LIN {X 0,Y 541.507,Z 325.44,A -85,B 0,C 180,E1 25518.834,E2 25518.834} C_VEL
LIN {X 0,Y 542.9,Z 340.233,A -85,B 0,C 180,E1 25517.69,E2 25517.69} C_VEL
LIN {X 0,Y 545.785,Z 352.594,A -85,B 0,C 180,E1 25516.608,E2 25516.608} C_VEL
LIN {X 0,Y 549.602,Z 361.822,A -85,B 0,C 180,E1 25515.687,E2 25515.687} C_VEL
LIN {X 0,Y 554.796,Z 369.914,A -85,B 0,C 180,E1 25514.76,E2 25514.76} C_VEL
LIN {X 0,Y 561.405,Z 376.773,A -85,B 0,C 180,E1 25513.838,E2 25513.838} C_VEL
LIN {X 0,Y 569.472,Z 382.283,A -85,B 0,C 180,E1 25512.933,E2 25512.933} C_VEL
LIN {X 0,Y 575.782,Z 385.075,A -85,B 0,C 180,E1 25512.29,E2 25512.29} C_VEL
LIN {X 0,Y 579.36,Z 385.747,A -85,B 0,C 180,E1 25511.772,E2 25511.772} C_VEL
LIN {X 0,Y 581.974,Z 385.283,A -85,B 0,C 180,E1 25511.193,E2 25511.193} C_VEL
LIN {X 0,Y 583.328,Z 383.79,A -85,B 0,C 180,E1 25510.595,E2 25510.595} C_VEL
LIN {X 0,Y 583.299,Z 381.198,A -85,B 0,C 180,E1 25509.985,E2 25509.985} C_VEL
LIN {X 0,Y 581.736,Z 377.706,A -85,B 0,C 180,E1 25509.426,E2 25509.426} C_VEL
LIN {X 0,Y 578.601,Z 373.318,A -85,B 0,C 180,E1 25508.946,E2 25508.946} C_VEL
LIN {X 0,Y 572.524,Z 363.934,A -85,B 0,C 180,E1 25508.187,E2 25508.187} C_VEL
LIN {X 0,Y 567.538,Z 353.434,A -85,B 0,C 180,E1 25507.542,E2 25507.542} C_VEL
LIN {X 0,Y 563.487,Z 341.539,A -85,B 0,C 180,E1 25507.003,E2 25507.003} C_VEL
LIN {X 0,Y 562.249,Z 337.195,A -85,B 0,C 180,E1 25506.836,E2 25506.836} C_VEL
LIN {X 0,Y 557.951,Z 382.113,A -85,B 0,C 180,E1 25506.242,E2 25506.242} C_VEL
LIN {X 0,Y 554.59,Z 408.363,A -85,B 0,C 180,E1 25505.766,E2 25505.766} C_VEL
LIN {X 0,Y 552.443,Z 419.215,A -85,B 0,C 180,E1 25505.456,E2 25505.456} C_VEL
LIN {X 0,Y 551.439,Z 422.72,A -85,B 0,C 180,E1 25505.309,E2 25505.309} C_VEL
LIN {X 0,Y 547.112,Z 475.176,A -85,B 0,C 180,E1 25504.664,E2 25504.664} C_VEL
LIN {X 0,Y 544.575,Z 495.316,A -85,B 0,C 180,E1 25504.346,E2 25504.346} C_VEL
LIN {X 0,Y 541.642,Z 509.391,A -85,B 0,C 180,E1 25504.002,E2 25504.002} C_VEL
LIN {X 0,Y 539.647,Z 516.391,A -85,B 0,C 180,E1 25503.689,E2 25503.689} C_VEL
LIN {X 0,Y 538.533,Z 609.219,A -85,B 0,C 180,E1 25502.262,E2 25502.262} C_VEL
LIN {X 0,Y 537.892,Z 631.012,A -85,B 0,C 180,E1 25501.735,E2 25501.735} C_VEL
LIN {X 0,Y 537.114,Z 653.311,A -85,B 0,C 180,E1 25500.979,E2 25500.979} C_VEL
LIN {X 0,Y 536.157,Z 674.428,A -85,B 0,C 180,E1 25500.054,E2 25500.054} C_VEL
LIN {X 0,Y 535.132,Z 694.792,A -85,B 0,C 180,E1 25498.942,E2 25498.942} C_VEL
LIN {X 0,Y 534.004,Z 714.986,A -85,B 0,C 180,E1 25497.608,E2 25497.608} C_VEL
LIN {X 0,Y 532.851,Z 734.82,A -85,B 0,C 180,E1 25496.046,E2 25496.046} C_VEL
LIN {X 0,Y 531.811,Z 752.831,A -85,B 0,C 180,E1 25494.374,E2 25494.374} C_VEL
LIN {X 0,Y 530.82,Z 770.22,A -85,B 0,C 180,E1 25492.481,E2 25492.481} C_VEL
LIN {X 0,Y 529.957,Z 786.287,A -85,B 0,C 180,E1 25490.428,E2 25490.428} C_VEL
LIN {X 0,Y 529.266,Z 800.604,A -85,B 0,C 180,E1 25488.276,E2 25488.276} C_VEL
LIN {X 0,Y 528.733,Z 813.274,A -85,B 0,C 180,E1 25486.027,E2 25486.027} C_VEL
LIN {X 0,Y 528.362,Z 824.318,A -85,B 0,C 180,E1 25483.683,E2 25483.683} C_VEL
LIN {X 0,Y 528.131,Z 833.313,A -85,B 0,C 180,E1 25481.355,E2 25481.355} C_VEL
LIN {X 0,Y 528.003,Z 840.399,A -85,B 0,C 180,E1 25479.043,E2 25479.043} C_VEL
LIN {X 0,Y 527.934,Z 846.011,A -85,B 0,C 180,E1 25476.634,E2 25476.634} C_VEL
LIN {X 0,Y 527.917,Z 849.739,A -85,B 0,C 180,E1 25474.345,E2 25474.345} C_VEL
LIN {X 0,Y 527.909,Z 851.902,A -85,B 0,C 180,E1 25471.954,E2 25471.954} C_VEL
LIN {X 0,Y 527.898,Z 852.445,A -85,B 0,C 180,E1 25469.566,E2 25469.566} C_VEL
LIN {X 0,Y 527.91,Z 851.331,A -85,B 0,C 180,E1 25467.177,E2 25467.177} C_VEL
LIN {X 0,Y 527.923,Z 848.489,A -85,B 0,C 180,E1 25464.784,E2 25464.784} C_VEL
LIN {X 0,Y 527.955,Z 843.939,A -85,B 0,C 180,E1 25462.382,E2 25462.382} C_VEL
LIN {X 0,Y 528.035,Z 837.923,A -85,B 0,C 180,E1 25460.078,E2 25460.078} C_VEL
LIN {X 0,Y 528.2,Z 830.099,A -85,B 0,C 180,E1 25457.76,E2 25457.76} C_VEL
LIN {X 0,Y 528.485,Z 820.356,A -85,B 0,C 180,E1 25455.426,E2 25455.426} C_VEL
LIN {X 0,Y 528.903,Z 809.121,A -85,B 0,C 180,E1 25453.188,E2 25453.188} C_VEL
LIN {X 0,Y 529.496,Z 795.627,A -85,B 0,C 180,E1 25450.932,E2 25450.932} C_VEL
LIN {X 0,Y 530.266,Z 780.344,A -85,B 0,C 180,E1 25448.775,E2 25448.775} C_VEL
LIN {X 0,Y 531.183,Z 763.692,A -85,B 0,C 180,E1 25446.774,E2 25446.774} C_VEL
LIN {X 0,Y 532.215,Z 745.663,A -85,B 0,C 180,E1 25444.929,E2 25444.929} C_VEL
LIN {X 0,Y 533.303,Z 727.139,A -85,B 0,C 180,E1 25443.319,E2 25443.319} C_VEL
LIN {X 0,Y 534.441,Z 707.515,A -85,B 0,C 180,E1 25441.871,E2 25441.871} C_VEL
LIN {X 0,Y 535.472,Z 687.857,A -85,B 0,C 180,E1 25440.655,E2 25440.655} C_VEL
LIN {X 0,Y 536.509,Z 667.145,A -85,B 0,C 180,E1 25439.603,E2 25439.603} C_VEL
LIN {X 0,Y 537.398,Z 645.684,A -85,B 0,C 180,E1 25438.736,E2 25438.736} C_VEL
LIN {X 0,Y 538.141,Z 623.996,A -85,B 0,C 180,E1 25438.074,E2 25438.074} C_VEL
LIN {X 0,Y 538.654,Z 601.949,A -85,B 0,C 180,E1 25437.607,E2 25437.607} C_VEL
LIN {X 0,Y 539.603,Z 521.674,A -85,B 0,C 180,E1 25436.387,E2 25436.387} C_VEL
LIN {X 0,Y 541.451,Z 515.855,A -85,B 0,C 180,E1 25436.104,E2 25436.104} C_VEL
LIN {X 0,Y 544.043,Z 503.404,A -85,B 0,C 180,E1 25435.787,E2 25435.787} C_VEL
LIN {X 0,Y 547.469,Z 471.343,A -85,B 0,C 180,E1 25435.282,E2 25435.282} C_VEL
LIN {X 0,Y 551.647,Z 421.541,A -85,B 0,C 180,E1 25434.661,E2 25434.661} C_VEL
LIN {X 0,Y 553.46,Z 414.673,A -85,B 0,C 180,E1 25434.397,E2 25434.397} C_VEL
LIN {X 0,Y 556.22,Z 396.703,A -85,B 0,C 180,E1 25434.002,E2 25434.002} C_VEL
LIN {X 0,Y 559.935,Z 363.496,A -85,B 0,C 180,E1 25433.482,E2 25433.482} C_VEL
LIN {X 0,Y 562.811,Z 376.767,A -85,B 0,C 180,E1 25433.088,E2 25433.088} C_VEL
LIN {X 0,Y 566.701,Z 388.825,A -85,B 0,C 180,E1 25432.568,E2 25432.568} C_VEL
LIN {X 0,Y 571.599,Z 399.681,A -85,B 0,C 180,E1 25431.931,E2 25431.931} C_VEL
LIN {X 0,Y 577.324,Z 409.005,A -85,B 0,C 180,E1 25431.206,E2 25431.206} C_VEL
LIN {X 0,Y 579.654,Z 413.297,A -85,B 0,C 180,E1 25430.724,E2 25430.724} C_VEL
LIN {X 0,Y 580.529,Z 416.774,A -85,B 0,C 180,E1 25430.155,E2 25430.155} C_VEL
LIN {X 0,Y 580.022,Z 419.104,A -85,B 0,C 180,E1 25429.597,E2 25429.597} C_VEL
LIN {X 0,Y 578.027,Z 420.583,A -85,B 0,C 180,E1 25428.954,E2 25428.954} C_VEL
LIN {X 0,Y 574.752,Z 420.735,A -85,B 0,C 180,E1 25428.352,E2 25428.352} C_VEL
LIN {X 0,Y 570.602,Z 419.567,A -85,B 0,C 180,E1 25427.835,E2 25427.835} C_VEL
LIN {X 0,Y 562.188,Z 414.887,A -85,B 0,C 180,E1 25426.967,E2 25426.967} C_VEL
LIN {X 0,Y 554.609,Z 408.372,A -85,B 0,C 180,E1 25425.998,E2 25425.998} C_VEL
LIN {X 0,Y 548.567,Z 400.431,A -85,B 0,C 180,E1 25424.992,E2 25424.992} C_VEL
LIN {X 0,Y 543.999,Z 390.85,A -85,B 0,C 180,E1 25423.934,E2 25423.934} C_VEL
LIN {X 0,Y 540.909,Z 379.13,A -85,B 0,C 180,E1 25422.79,E2 25422.79} C_VEL
LIN {X 0,Y 539.455,Z 365.314,A -85,B 0,C 180,E1 25421.57,E2 25421.57} C_VEL
LIN {X 0,Y 540.181,Z 339.074,A -85,B 0,C 180,E1 25419.479,E2 25419.479} C_VEL
LIN {X 0,Y 542.247,Z 299.859,A -85,B 0,C 180,E1 25416.312,E2 25416.312} C_VEL
LIN {X 0,Y 543.435,Z 278.465,A -85,B 0,C 180,E1 25414.519,E2 25414.519} C_VEL
LIN {X 0,Y 536.159,Z 263.024,A -85,B 0,C 180,E1 25412.232,E2 25412.232} C_VEL
LIN {X 0,Y 532.304,Z 255.135,A -85,B 0,C 180,E1 25410.975,E2 25410.975} C_VEL
LIN {X 0,Y 530.079,Z 250.727,A -85,B 0,C 180,E1 25410.24,E2 25410.24} C_VEL
LIN {X 0,Y 528.598,Z 247.484,A -85,B 0,C 180,E1 25409.708,E2 25409.708} C_VEL
LIN {X 0,Y 528.503,Z 246.905,A -85,B 0,C 180,E1 25409.589,E2 25409.589} C_VEL
LIN {X 0,Y 528.518,Z 247.111,A -85,B 0,C 180,E1 25407.776,E2 25407.776} C_VEL
LIN {X 0,Y 530.21,Z 254.424,A -85,B 0,C 180,E1 25407.274,E2 25407.274} C_VEL
LIN {X 0,Y 530.852,Z 299.671,A -85,B 0,C 180,E1 25404.42,E2 25404.42} C_VEL
LIN {X 0,Y 531.29,Z 341.245,A -85,B 0,C 180,E1 25401.645,E2 25401.645} C_VEL
LIN {X 0,Y 531.277,Z 383.369,A -85,B 0,C 180,E1 25398.716,E2 25398.716} C_VEL
LIN {X 0,Y 530.854,Z 431.931,A -85,B 0,C 180,E1 25395.233,E2 25395.233} C_VEL
LIN {X 0,Y 530.24,Z 479.348,A -85,B 0,C 180,E1 25391.75,E2 25391.75} C_VEL
LIN {X 0,Y 530.109,Z 491.534,A -85,B 0,C 180,E1 25390.885,E2 25390.885} C_VEL
LIN {X 0,Y 529.689,Z 604.749,A -85,B 0,C 180,E1 25389.291,E2 25389.291} C_VEL
LIN {X 0,Y 529.568,Z 619.615,A -85,B 0,C 180,E1 25388.872,E2 25388.872} C_VEL
LIN {X 0,Y 529.421,Z 632.902,A -85,B 0,C 180,E1 25388.307,E2 25388.307} C_VEL
LIN {X 0,Y 529.2,Z 645.983,A -85,B 0,C 180,E1 25387.545,E2 25387.545} C_VEL
LIN {X 0,Y 528.96,Z 658.621,A -85,B 0,C 180,E1 25386.566,E2 25386.566} C_VEL
LIN {X 0,Y 528.737,Z 669.029,A -85,B 0,C 180,E1 25385.534,E2 25385.534} C_VEL
LIN {X 0,Y 528.525,Z 678.575,A -85,B 0,C 180,E1 25384.339,E2 25384.339} C_VEL
LIN {X 0,Y 528.346,Z 687.273,A -85,B 0,C 180,E1 25382.928,E2 25382.928} C_VEL
LIN {X 0,Y 528.206,Z 693.851,A -85,B 0,C 180,E1 25381.518,E2 25381.518} C_VEL
LIN {X 0,Y 528.13,Z 699.006,A -85,B 0,C 180,E1 25380,E2 25380} C_VEL
LIN {X 0,Y 528.078,Z 702.566,A -85,B 0,C 180,E1 25378.372,E2 25378.372} C_VEL
LIN {X 0,Y 528.064,Z 704.318,A -85,B 0,C 180,E1 25376.635,E2 25376.635} C_VEL
LIN {X 0,Y 528.051,Z 704.126,A -85,B 0,C 180,E1 25375.003,E2 25375.003} C_VEL
LIN {X 0,Y 528.068,Z 702.145,A -85,B 0,C 180,E1 25373.367,E2 25373.367} C_VEL
LIN {X 0,Y 528.104,Z 698.628,A -85,B 0,C 180,E1 25371.836,E2 25371.836} C_VEL
LIN {X 0,Y 528.191,Z 692.798,A -85,B 0,C 180,E1 25370.19,E2 25370.19} C_VEL
LIN {X 0,Y 528.319,Z 685.733,A -85,B 0,C 180,E1 25368.759,E2 25368.759} C_VEL
LIN {X 0,Y 528.492,Z 677.206,A -85,B 0,C 180,E1 25367.433,E2 25367.433} C_VEL
LIN {X 0,Y 528.72,Z 667.179,A -85,B 0,C 180,E1 25366.215,E2 25366.215} C_VEL
LIN {X 0,Y 528.965,Z 655.414,A -85,B 0,C 180,E1 25365.103,E2 25365.103} C_VEL
LIN {X 0,Y 529.203,Z 643.22,A -85,B 0,C 180,E1 25364.212,E2 25364.212} C_VEL
LIN {X 0,Y 529.426,Z 630.244,A -85,B 0,C 180,E1 25363.487,E2 25363.487} C_VEL
LIN {X 0,Y 529.616,Z 615.198,A -85,B 0,C 180,E1 25362.889,E2 25362.889} C_VEL
LIN {X 0,Y 529.731,Z 599.229,A -85,B 0,C 180,E1 25362.502,E2 25362.502} C_VEL
LIN {X 0,Y 529.967,Z 489.753,A -85,B 0,C 180,E1 25360.978,E2 25360.978} C_VEL
LIN {X 0,Y 529.944,Z 486.878,A -85,B 0,C 180,E1 25360.802,E2 25360.802} C_VEL
LIN {X 0,Y 530.358,Z 460.271,A -85,B 0,C 180,E1 25358.814,E2 25358.814} C_VEL
LIN {X 0,Y 529.49,Z 454.16,A -85,B 0,C 180,E1 25358.319,E2 25358.319} C_VEL
LIN {X 0,Y 523.776,Z 438.358,A -85,B 0,C 180,E1 25356.901,E2 25356.901} C_VEL
LIN {X 0,Y 523.166,Z 432.941,A -85,B 0,C 180,E1 25356.467,E2 25356.467} C_VEL
LIN {X 0,Y 523.904,Z 387.135,A -85,B 0,C 180,E1 25353.033,E2 25353.033} C_VEL
LIN {X 0,Y 524.522,Z 341.101,A -85,B 0,C 180,E1 25349.595,E2 25349.595} C_VEL
LIN {X 0,Y 524.914,Z 297.566,A -85,B 0,C 180,E1 25346.337,E2 25346.337} C_VEL
LIN {X 0,Y 525.147,Z 262.725,A -85,B 0,C 180,E1 25343.739,E2 25343.739} C_VEL
LIN {X 0,Y 520.574,Z 247.885,A -85,B 0,C 180,E1 25342.354,E2 25342.354} C_VEL
LIN {X 0,Y 520.575,Z 247.892,A -85,B 0,C 180,E1 25338.791,E2 25338.791} C_VEL
LIN {X 0,Y 520.564,Z 247.895,A -85,B 0,C 180,E1 25335.446,E2 25335.446} C_VEL
LIN {X 0,Y 520.591,Z 247.964,A -85,B 0,C 180,E1 25333.248,E2 25333.248} C_VEL
LIN {X 0,Y 521.88,Z 251.385,A -85,B 0,C 180,E1 25332.633,E2 25332.633} C_VEL
LIN {X 0,Y 524.834,Z 257.768,A -85,B 0,C 180,E1 25331.439,E2 25331.439} C_VEL
LIN {X 0,Y 530.138,Z 269.708,A -85,B 0,C 180,E1 25329.325,E2 25329.325} C_VEL
LIN {X 0,Y 532.076,Z 275.112,A -85,B 0,C 180,E1 25328.463,E2 25328.463} C_VEL
LIN {X 0,Y 529.458,Z 306.929,A -85,B 0,C 180,E1 25325.183,E2 25325.183} C_VEL
LIN {X 0,Y 531.569,Z 317.62,A -85,B 0,C 180,E1 25324.852,E2 25324.852} C_VEL
LIN {X 0,Y 528.989,Z 544.595,A -85,B 0,C 180,E1 25321.435,E2 25321.435} C_VEL
LIN {X 0,Y 528.578,Z 567.627,A -85,B 0,C 180,E1 25321.026,E2 25321.026} C_VEL
LIN {X 0,Y 527.977,Z 588.155,A -85,B 0,C 180,E1 25320.456,E2 25320.456} C_VEL
LIN {X 0,Y 527.322,Z 605.247,A -85,B 0,C 180,E1 25319.819,E2 25319.819} C_VEL
LIN {X 0,Y 526.551,Z 623.634,A -85,B 0,C 180,E1 25318.961,E2 25318.961} C_VEL
LIN {X 0,Y 525.565,Z 642.685,A -85,B 0,C 180,E1 25317.843,E2 25317.843} C_VEL
LIN {X 0,Y 524.73,Z 658.626,A -85,B 0,C 180,E1 25316.724,E2 25316.724} C_VEL
LIN {X 0,Y 523.753,Z 676.293,A -85,B 0,C 180,E1 25315.257,E2 25315.257} C_VEL
LIN {X 0,Y 522.9,Z 691.093,A -85,B 0,C 180,E1 25313.795,E2 25313.795} C_VEL
LIN {X 0,Y 522.144,Z 705.392,A -85,B 0,C 180,E1 25312.163,E2 25312.163} C_VEL
LIN {X 0,Y 521.439,Z 719.102,A -85,B 0,C 180,E1 25310.308,E2 25310.308} C_VEL
LIN {X 0,Y 520.919,Z 730.743,A -85,B 0,C 180,E1 25308.464,E2 25308.464} C_VEL
LIN {X 0,Y 520.481,Z 742.217,A -85,B 0,C 180,E1 25306.288,E2 25306.288} C_VEL
LIN {X 0,Y 520.219,Z 750.632,A -85,B 0,C 180,E1 25304.356,E2 25304.356} C_VEL
LIN {X 0,Y 520.054,Z 758.283,A -85,B 0,C 180,E1 25302.21,E2 25302.21} C_VEL
LIN {X 0,Y 519.961,Z 764.345,A -85,B 0,C 180,E1 25299.966,E2 25299.966} C_VEL
LIN {X 0,Y 519.929,Z 768.375,A -85,B 0,C 180,E1 25297.95,E2 25297.95} C_VEL
LIN {X 0,Y 519.907,Z 771.321,A -85,B 0,C 180,E1 25295.629,E2 25295.629} C_VEL
LIN {X 0,Y 519.903,Z 772.378,A -85,B 0,C 180,E1 25293.503,E2 25293.503} C_VEL
LIN {X 0,Y 519.903,Z 772.051,A -85,B 0,C 180,E1 25291.322,E2 25291.322} C_VEL
LIN {X 0,Y 519.918,Z 769.904,A -85,B 0,C 180,E1 25289.008,E2 25289.008} C_VEL
LIN {X 0,Y 519.938,Z 766.672,A -85,B 0,C 180,E1 25287.024,E2 25287.024} C_VEL
LIN {X 0,Y 519.998,Z 761.549,A -85,B 0,C 180,E1 25284.815,E2 25284.815} C_VEL
LIN {X 0,Y 520.128,Z 754.549,A -85,B 0,C 180,E1 25282.6,E2 25282.6} C_VEL
LIN {X 0,Y 520.317,Z 747.153,A -85,B 0,C 180,E1 25280.711,E2 25280.711} C_VEL
LIN {X 0,Y 520.674,Z 737.117,A -85,B 0,C 180,E1 25278.592,E2 25278.592} C_VEL
LIN {X 0,Y 521.109,Z 726.154,A -85,B 0,C 180,E1 25276.688,E2 25276.688} C_VEL
LIN {X 0,Y 521.687,Z 714.146,A -85,B 0,C 180,E1 25274.891,E2 25274.891} C_VEL
LIN {X 0,Y 522.451,Z 699.354,A -85,B 0,C 180,E1 25273.031,E2 25273.031} C_VEL
LIN {X 0,Y 523.195,Z 685.995,A -85,B 0,C 180,E1 25271.588,E2 25271.588} C_VEL
LIN {X 0,Y 524.155,Z 669.279,A -85,B 0,C 180,E1 25270.034,E2 25270.034} C_VEL
LIN {X 0,Y 525.053,Z 652.42,A -85,B 0,C 180,E1 25268.729,E2 25268.729} C_VEL
LIN {X 0,Y 525.934,Z 636.075,A -85,B 0,C 180,E1 25267.652,E2 25267.652} C_VEL
LIN {X 0,Y 526.869,Z 616.032,A -85,B 0,C 180,E1 25266.573,E2 25266.573} C_VEL
LIN {X 0,Y 527.585,Z 598.852,A -85,B 0,C 180,E1 25265.836,E2 25265.836} C_VEL
LIN {X 0,Y 528.241,Z 580.125,A -85,B 0,C 180,E1 25265.201,E2 25265.201} C_VEL
LIN {X 0,Y 528.768,Z 559.287,A -85,B 0,C 180,E1 25264.715,E2 25264.715} C_VEL
LIN {X 0,Y 531.644,Z 314.439,A -85,B 0,C 180,E1 25261.011,E2 25261.011} C_VEL
LIN {X 0,Y 529.934,Z 304.934,A -85,B 0,C 180,E1 25260.716,E2 25260.716} C_VEL
LIN {X 0,Y 532.112,Z 274.325,A -85,B 0,C 180,E1 25258.065,E2 25258.065} C_VEL
LIN {X 0,Y 529.618,Z 267.665,A -85,B 0,C 180,E1 25257.153,E2 25257.153} C_VEL
LIN {X 0,Y 523.77,Z 255.31,A -85,B 0,C 180,E1 25255.267,E2 25255.267} C_VEL
LIN {X 0,Y 522.007,Z 251.554,A -85,B 0,C 180,E1 25254.684,E2 25254.684} C_VEL
LIN {X 0,Y 520.594,Z 247.941,A -85,B 0,C 180,E1 25254.153,E2 25254.153} C_VEL
LIN {X 0,Y 520.583,Z 247.897,A -85,B 0,C 180,E1 25250.667,E2 25250.667} C_VEL
LIN {X 0,Y 520.576,Z 247.893,A -85,B 0,C 180,E1 25247.162,E2 25247.162} C_VEL
LIN {X 0,Y 520.585,Z 247.89,A -85,B 0,C 180,E1 25243.592,E2 25243.592} C_VEL
LIN {X 0,Y 520.589,Z 247.883,A -85,B 0,C 180,E1 25239.974,E2 25239.974} C_VEL
LIN {X 0,Y 520.57,Z 247.88,A -85,B 0,C 180,E1 25236.543,E2 25236.543} C_VEL
LIN {X 0,Y 520.567,Z 247.893,A -85,B 0,C 180,E1 25233.13,E2 25233.13} C_VEL
LIN {X 0,Y 520.582,Z 247.891,A -85,B 0,C 180,E1 25229.705,E2 25229.705} C_VEL
LIN {X 0,Y 520.591,Z 247.925,A -85,B 0,C 180,E1 25229.168,E2 25229.168} C_VEL
LIN {X 0,Y 525.449,Z 263.917,A -85,B 0,C 180,E1 25227.604,E2 25227.604} C_VEL
LIN {X 0,Y 525.069,Z 309.421,A -85,B 0,C 180,E1 25223.929,E2 25223.929} C_VEL
LIN {X 0,Y 524.544,Z 350.281,A -85,B 0,C 180,E1 25220.622,E2 25220.622} C_VEL
LIN {X 0,Y 523.837,Z 391.693,A -85,B 0,C 180,E1 25217.266,E2 25217.266} C_VEL
LIN {X 0,Y 523.058,Z 434.806,A -85,B 0,C 180,E1 25213.774,E2 25213.774} C_VEL
LIN {X 0,Y 523.011,Z 441.178,A -85,B 0,C 180,E1 25213.284,E2 25213.284} C_VEL
LIN {X 0,Y 523.43,Z 448.653,A -85,B 0,C 180,E1 25213.159,E2 25213.159} C_VEL
LIN {X 0,Y 522.655,Z 583.279,A -85,B 0,C 180,E1 25211.221,E2 25211.221} C_VEL
LIN {X 0,Y 522.498,Z 600.137,A -85,B 0,C 180,E1 25210.764,E2 25210.764} C_VEL
LIN {X 0,Y 522.241,Z 615.223,A -85,B 0,C 180,E1 25210.145,E2 25210.145} C_VEL
LIN {X 0,Y 521.93,Z 630.251,A -85,B 0,C 180,E1 25209.316,E2 25209.316} C_VEL
LIN {X 0,Y 521.561,Z 643.994,A -85,B 0,C 180,E1 25208.322,E2 25208.322} C_VEL
LIN {X 0,Y 521.215,Z 656.762,A -85,B 0,C 180,E1 25207.163,E2 25207.163} C_VEL
LIN {X 0,Y 520.87,Z 668.3,A -85,B 0,C 180,E1 25205.84,E2 25205.84} C_VEL
LIN {X 0,Y 520.592,Z 678.338,A -85,B 0,C 180,E1 25204.406,E2 25204.406} C_VEL
LIN {X 0,Y 520.364,Z 687.336,A -85,B 0,C 180,E1 25202.754,E2 25202.754} C_VEL
LIN {X 0,Y 520.235,Z 694.19,A -85,B 0,C 180,E1 25201.102,E2 25201.102} C_VEL
LIN {X 0,Y 520.145,Z 699.485,A -85,B 0,C 180,E1 25199.34,E2 25199.34} C_VEL
LIN {X 0,Y 520.109,Z 702.89,A -85,B 0,C 180,E1 25197.576,E2 25197.576} C_VEL
LIN {X 0,Y 520.09,Z 704.669,A -85,B 0,C 180,E1 25195.701,E2 25195.701} C_VEL
LIN {X 0,Y 520.109,Z 704.494,A -85,B 0,C 180,E1 25193.82,E2 25193.82} C_VEL
LIN {X 0,Y 520.131,Z 702.635,A -85,B 0,C 180,E1 25192.045,E2 25192.045} C_VEL
LIN {X 0,Y 520.214,Z 698.662,A -85,B 0,C 180,E1 25190.151,E2 25190.151} C_VEL
LIN {X 0,Y 520.308,Z 693.317,A -85,B 0,C 180,E1 25188.472,E2 25188.472} C_VEL
LIN {X 0,Y 520.48,Z 685.988,A -85,B 0,C 180,E1 25186.786,E2 25186.786} C_VEL
LIN {X 0,Y 520.703,Z 677.667,A -85,B 0,C 180,E1 25185.318,E2 25185.318} C_VEL
LIN {X 0,Y 521.01,Z 667.107,A -85,B 0,C 180,E1 25183.844,E2 25183.844} C_VEL
LIN {X 0,Y 521.348,Z 655.434,A -85,B 0,C 180,E1 25182.561,E2 25182.561} C_VEL
LIN {X 0,Y 521.672,Z 642.791,A -85,B 0,C 180,E1 25181.449,E2 25181.449} C_VEL
LIN {X 0,Y 521.978,Z 629.493,A -85,B 0,C 180,E1 25180.531,E2 25180.531} C_VEL
LIN {X 0,Y 522.256,Z 614.349,A -85,B 0,C 180,E1 25179.725,E2 25179.725} C_VEL
LIN {X 0,Y 522.446,Z 598.144,A -85,B 0,C 180,E1 25179.115,E2 25179.115} C_VEL
LIN {X 0,Y 522.534,Z 582.01,A -85,B 0,C 180,E1 25178.721,E2 25178.721} C_VEL
LIN {X 0,Y 523.158,Z 443.793,A -85,B 0,C 180,E1 25176.748,E2 25176.748} C_VEL
LIN {X 0,Y 523.672,Z 404.384,A -85,B 0,C 180,E1 25173.646,E2 25173.646} C_VEL
LIN {X 0,Y 523.889,Z 371.931,A -85,B 0,C 180,E1 25171.166,E2 25171.166} C_VEL
LIN {X 0,Y 523.796,Z 336.608,A -85,B 0,C 180,E1 25168.569,E2 25168.569} C_VEL
LIN {X 0,Y 523.55,Z 314.757,A -85,B 0,C 180,E1 25167.025,E2 25167.025} C_VEL
LIN {X 0,Y 523.146,Z 296.005,A -85,B 0,C 180,E1 25165.747,E2 25165.747} C_VEL
LIN {X 0,Y 522.577,Z 275.208,A -85,B 0,C 180,E1 25164.366,E2 25164.366} C_VEL
LIN {X 0,Y 523.902,Z 276.373,A -85,B 0,C 180,E1 25164.133,E2 25164.133} C_VEL
LIN {X 0,Y 526.059,Z 276.444,A -85,B 0,C 180,E1 25163.9,E2 25163.9} C_VEL
LIN {X 0,Y 528.145,Z 275.832,A -85,B 0,C 180,E1 25163.729,E2 25163.729} C_VEL
LIN {X 0,Y 532.182,Z 275.841,A -85,B 0,C 180,E1 25163.313,E2 25163.313} C_VEL
LIN {X 0,Y 534.075,Z 275.725,A -85,B 0,C 180,E1 25163.129,E2 25163.129} C_VEL
LIN {X 0,Y 536.509,Z 281.057,A -85,B 0,C 180,E1 25162.487,E2 25162.487} C_VEL
LIN {X 0,Y 534.887,Z 327.338,A -85,B 0,C 180,E1 25159.279,E2 25159.279} C_VEL
LIN {X 0,Y 536.19,Z 342.822,A -85,B 0,C 180,E1 25158.077,E2 25158.077} C_VEL
LIN {X 0,Y 539.016,Z 355.68,A -85,B 0,C 180,E1 25156.951,E2 25156.951} C_VEL
LIN {X 0,Y 543.144,Z 366.122,A -85,B 0,C 180,E1 25155.905,E2 25155.905} C_VEL
LIN {X 0,Y 548.239,Z 374.394,A -85,B 0,C 180,E1 25154.959,E2 25154.959} C_VEL
LIN {X 0,Y 554.714,Z 381.547,A -85,B 0,C 180,E1 25154.013,E2 25154.013} C_VEL
LIN {X 0,Y 562.613,Z 387.469,A -85,B 0,C 180,E1 25153.079,E2 25153.079} C_VEL
LIN {X 0,Y 571.91,Z 391.956,A -85,B 0,C 180,E1 25152.161,E2 25152.161} C_VEL
LIN {X 0,Y 575.707,Z 392.866,A -85,B 0,C 180,E1 25151.686,E2 25151.686} C_VEL
LIN {X 0,Y 578.745,Z 392.728,A -85,B 0,C 180,E1 25151.128,E2 25151.128} C_VEL
LIN {X 0,Y 580.519,Z 391.66,A -85,B 0,C 180,E1 25150.575,E2 25150.575} C_VEL
LIN {X 0,Y 581.132,Z 389.511,A -85,B 0,C 180,E1 25149.959,E2 25149.959} C_VEL
LIN {X 0,Y 580.198,Z 386.328,A -85,B 0,C 180,E1 25149.359,E2 25149.359} C_VEL
LIN {X 0,Y 577.776,Z 382.509,A -85,B 0,C 180,E1 25148.853,E2 25148.853} C_VEL
LIN {X 0,Y 571.213,Z 373.317,A -85,B 0,C 180,E1 25148.02,E2 25148.02} C_VEL
LIN {X 0,Y 565.562,Z 362.684,A -85,B 0,C 180,E1 25147.282,E2 25147.282} C_VEL
LIN {X 0,Y 564.939,Z 361.378,A -85,B 0,C 180,E1 25147.198,E2 25147.198} C_VEL
LIN {X 0,Y 560.884,Z 398.192,A -85,B 0,C 180,E1 25146.649,E2 25146.649} C_VEL
LIN {X 0,Y 558.007,Z 416.875,A -85,B 0,C 180,E1 25146.25,E2 25146.25} C_VEL
LIN {X 0,Y 555.908,Z 425.833,A -85,B 0,C 180,E1 25145.954,E2 25145.954} C_VEL
LIN {X 0,Y 552.122,Z 468.82,A -85,B 0,C 180,E1 25145.459,E2 25145.459} C_VEL
LIN {X 0,Y 548.349,Z 490.191,A -85,B 0,C 180,E1 25145.233,E2 25145.233} C_VEL
LIN {X 0,Y 544.101,Z 506.941,A -85,B 0,C 180,E1 25144.936,E2 25144.936} C_VEL
LIN {X 0,Y 541.094,Z 517.425,A -85,B 0,C 180,E1 25144.586,E2 25144.586} C_VEL
LIN {X 0,Y 540.19,Z 520.542,A -85,B 0,C 180,E1 25144.467,E2 25144.467} C_VEL
LIN {X 0,Y 536.242,Z 533.852,A -85,B 0,C 180,E1 25144.206,E2 25144.206} C_VEL
LIN {X 0,Y 533.281,Z 543.81,A -85,B 0,C 180,E1 25143.839,E2 25143.839} C_VEL
LIN {X 0,Y 532.536,Z 547.21,A -85,B 0,C 180,E1 25143.688,E2 25143.688} C_VEL
LIN {X 0,Y 531.764,Z 609.206,A -85,B 0,C 180,E1 25142.723,E2 25142.723} C_VEL
LIN {X 0,Y 531.068,Z 630.869,A -85,B 0,C 180,E1 25142.196,E2 25142.196} C_VEL
LIN {X 0,Y 530.202,Z 653.306,A -85,B 0,C 180,E1 25141.428,E2 25141.428} C_VEL
LIN {X 0,Y 529.151,Z 674.305,A -85,B 0,C 180,E1 25140.5,E2 25140.5} C_VEL
LIN {X 0,Y 528.008,Z 694.799,A -85,B 0,C 180,E1 25139.371,E2 25139.371} C_VEL
LIN {X 0,Y 526.77,Z 714.714,A -85,B 0,C 180,E1 25138.041,E2 25138.041} C_VEL
LIN {X 0,Y 525.528,Z 734.139,A -85,B 0,C 180,E1 25136.497,E2 25136.497} C_VEL
LIN {X 0,Y 524.353,Z 752.271,A -85,B 0,C 180,E1 25134.804,E2 25134.804} C_VEL
LIN {X 0,Y 523.196,Z 770.219,A -85,B 0,C 180,E1 25132.827,E2 25132.827} C_VEL
LIN {X 0,Y 522.228,Z 786.289,A -85,B 0,C 180,E1 25130.745,E2 25130.745} C_VEL
LIN {X 0,Y 521.448,Z 800.607,A -85,B 0,C 180,E1 25128.56,E2 25128.56} C_VEL
LIN {X 0,Y 520.844,Z 813.278,A -85,B 0,C 180,E1 25126.277,E2 25126.277} C_VEL
LIN {X 0,Y 520.423,Z 824.321,A -85,B 0,C 180,E1 25123.896,E2 25123.896} C_VEL
LIN {X 0,Y 520.164,Z 833.312,A -85,B 0,C 180,E1 25121.532,E2 25121.532} C_VEL
LIN {X 0,Y 520.022,Z 840.402,A -85,B 0,C 180,E1 25119.183,E2 25119.183} C_VEL
LIN {X 0,Y 519.943,Z 846.012,A -85,B 0,C 180,E1 25116.737,E2 25116.737} C_VEL
LIN {X 0,Y 519.918,Z 849.739,A -85,B 0,C 180,E1 25114.412,E2 25114.412} C_VEL
LIN {X 0,Y 519.909,Z 851.904,A -85,B 0,C 180,E1 25111.984,E2 25111.984} C_VEL
LIN {X 0,Y 519.897,Z 852.447,A -85,B 0,C 180,E1 25109.559,E2 25109.559} C_VEL
LIN {X 0,Y 519.911,Z 851.33,A -85,B 0,C 180,E1 25107.134,E2 25107.134} C_VEL
LIN {X 0,Y 519.924,Z 848.491,A -85,B 0,C 180,E1 25104.704,E2 25104.704} C_VEL
LIN {X 0,Y 519.965,Z 843.942,A -85,B 0,C 180,E1 25102.264,E2 25102.264} C_VEL
LIN {X 0,Y 520.065,Z 837.703,A -85,B 0,C 180,E1 25099.849,E2 25099.849} C_VEL
LIN {X 0,Y 520.254,Z 829.859,A -85,B 0,C 180,E1 25097.502,E2 25097.502} C_VEL
LIN {X 0,Y 520.566,Z 820.359,A -85,B 0,C 180,E1 25095.199,E2 25095.199} C_VEL
LIN {X 0,Y 521.038,Z 809.122,A -85,B 0,C 180,E1 25092.926,E2 25092.926} C_VEL
LIN {X 0,Y 521.713,Z 795.628,A -85,B 0,C 180,E1 25090.637,E2 25090.637} C_VEL
LIN {X 0,Y 522.581,Z 780.347,A -85,B 0,C 180,E1 25088.447,E2 25088.447} C_VEL
LIN {X 0,Y 523.6,Z 763.826,A -85,B 0,C 180,E1 25086.433,E2 25086.433} C_VEL
LIN {X 0,Y 524.752,Z 745.949,A -85,B 0,C 180,E1 25084.575,E2 25084.575} C_VEL
LIN {X 0,Y 525.969,Z 727.143,A -85,B 0,C 180,E1 25082.916,E2 25082.916} C_VEL
LIN {X 0,Y 527.241,Z 707.51,A -85,B 0,C 180,E1 25081.452,E2 25081.452} C_VEL
LIN {X 0,Y 528.397,Z 687.754,A -85,B 0,C 180,E1 25080.217,E2 25080.217} C_VEL
LIN {X 0,Y 529.534,Z 667.155,A -85,B 0,C 180,E1 25079.16,E2 25079.16} C_VEL
LIN {X 0,Y 530.523,Z 645.582,A -85,B 0,C 180,E1 25078.28,E2 25078.28} C_VEL
LIN {X 0,Y 531.337,Z 623.823,A -85,B 0,C 180,E1 25077.611,E2 25077.611} C_VEL
LIN {X 0,Y 531.909,Z 601.529,A -85,B 0,C 180,E1 25077.138,E2 25077.138} C_VEL
LIN {X 0,Y 532.586,Z 549.761,A -85,B 0,C 180,E1 25076.338,E2 25076.338} C_VEL
LIN {X 0,Y 535.149,Z 542.227,A -85,B 0,C 180,E1 25075.973,E2 25075.973} C_VEL
LIN {X 0,Y 538.819,Z 531.538,A -85,B 0,C 180,E1 25075.695,E2 25075.695} C_VEL
LIN {X 0,Y 541.072,Z 524.39,A -85,B 0,C 180,E1 25075.574,E2 25075.574} C_VEL
LIN {X 0,Y 543.784,Z 516.045,A -85,B 0,C 180,E1 25075.249,E2 25075.249} C_VEL
LIN {X 0,Y 547.567,Z 502.172,A -85,B 0,C 180,E1 25074.979,E2 25074.979} C_VEL
LIN {X 0,Y 550.905,Z 483.263,A -85,B 0,C 180,E1 25074.753,E2 25074.753} C_VEL
LIN {X 0,Y 555.368,Z 432.966,A -85,B 0,C 180,E1 25074.123,E2 25074.123} C_VEL
LIN {X 0,Y 556.166,Z 424.2,A -85,B 0,C 180,E1 25074.009,E2 25074.009} C_VEL
LIN {X 0,Y 558.34,Z 414.988,A -85,B 0,C 180,E1 25073.703,E2 25073.703} C_VEL
LIN {X 0,Y 561.407,Z 394.031,A -85,B 0,C 180,E1 25073.279,E2 25073.279} C_VEL
LIN {X 0,Y 561.875,Z 391.087,A -85,B 0,C 180,E1 25073.215,E2 25073.215} C_VEL
LIN {X 0,Y 566.7,Z 402.577,A -85,B 0,C 180,E1 25072.568,E2 25072.568} C_VEL
LIN {X 0,Y 572.524,Z 412.796,A -85,B 0,C 180,E1 25071.813,E2 25071.813} C_VEL
LIN {X 0,Y 576.065,Z 418.186,A -85,B 0,C 180,E1 25071.297,E2 25071.297} C_VEL
LIN {X 0,Y 577.663,Z 422.07,A -85,B 0,C 180,E1 25070.755,E2 25070.755} C_VEL
LIN {X 0,Y 577.761,Z 424.939,A -85,B 0,C 180,E1 25070.184,E2 25070.184} C_VEL
LIN {X 0,Y 576.394,Z 426.951,A -85,B 0,C 180,E1 25069.551,E2 25069.551} C_VEL
LIN {X 0,Y 573.859,Z 427.759,A -85,B 0,C 180,E1 25068.976,E2 25068.976} C_VEL
LIN {X 0,Y 570.415,Z 427.444,A -85,B 0,C 180,E1 25068.458,E2 25068.458} C_VEL
LIN {X 0,Y 565.558,Z 425.733,A -85,B 0,C 180,E1 25067.947,E2 25067.947} C_VEL
LIN {X 0,Y 556.426,Z 420.495,A -85,B 0,C 180,E1 25066.999,E2 25066.999} C_VEL
LIN {X 0,Y 548.86,Z 413.935,A -85,B 0,C 180,E1 25066.019,E2 25066.019} C_VEL
LIN {X 0,Y 542.318,Z 405.385,A -85,B 0,C 180,E1 25064.92,E2 25064.92} C_VEL
LIN {X 0,Y 537.481,Z 395.309,A -85,B 0,C 180,E1 25063.79,E2 25063.79} C_VEL
LIN {X 0,Y 534.246,Z 383.148,A -85,B 0,C 180,E1 25062.575,E2 25062.575} C_VEL
LIN {X 0,Y 532.752,Z 369.564,A -85,B 0,C 180,E1 25061.347,E2 25061.347} C_VEL
LIN {X 0,Y 533.19,Z 348.264,A -85,B 0,C 180,E1 25059.611,E2 25059.611} C_VEL
LIN {X 0,Y 535.529,Z 308.127,A -85,B 0,C 180,E1 25056.355,E2 25056.355} C_VEL
LIN {X 0,Y 537.107,Z 282.673,A -85,B 0,C 180,E1 25054.207,E2 25054.207} C_VEL
LIN {X 0,Y 530.236,Z 267.987,A -85,B 0,C 180,E1 25051.997,E2 25051.997} C_VEL
LIN {X 0,Y 524.536,Z 256.334,A -85,B 0,C 180,E1 25050.087,E2 25050.087} C_VEL
LIN {X 0,Y 522.366,Z 252.032,A -85,B 0,C 180,E1 25049.341,E2 25049.341} C_VEL
LIN {X 0,Y 520.822,Z 249.054,A -85,B 0,C 180,E1 25048.807,E2 25048.807} C_VEL
LIN {X 0,Y 520.587,Z 247.884,A -85,B 0,C 180,E1 25048.629,E2 25048.629} C_VEL
LIN {X 0,Y 520.596,Z 248.14,A -85,B 0,C 180,E1 25048.023,E2 25048.023} C_VEL
LIN {X 0,Y 522.581,Z 256.272,A -85,B 0,C 180,E1 25047.458,E2 25047.458} C_VEL
LIN {X 0,Y 523.216,Z 301.22,A -85,B 0,C 180,E1 25044.619,E2 25044.619} C_VEL
LIN {X 0,Y 523.655,Z 342.604,A -85,B 0,C 180,E1 25041.859,E2 25041.859} C_VEL
LIN {X 0,Y 523.601,Z 378.474,A -85,B 0,C 180,E1 25039.348,E2 25039.348} C_VEL
LIN {X 0,Y 523.344,Z 421.313,A -85,B 0,C 180,E1 25036.31,E2 25036.31} C_VEL
LIN {X 0,Y 522.791,Z 466.021,A -85,B 0,C 180,E1 25033.042,E2 25033.042} C_VEL
LIN {X 0,Y 522.395,Z 492.982,A -85,B 0,C 180,E1 25031.079,E2 25031.079} C_VEL
LIN {X 0,Y 521.867,Z 606.486,A -85,B 0,C 180,E1 25029.445,E2 25029.445} C_VEL
LIN {X 0,Y 521.762,Z 621.591,A -85,B 0,C 180,E1 25029.008,E2 25029.008} C_VEL
LIN {X 0,Y 521.621,Z 634.673,A -85,B 0,C 180,E1 25028.437,E2 25028.437} C_VEL
LIN {X 0,Y 521.395,Z 647.787,A -85,B 0,C 180,E1 25027.659,E2 25027.659} C_VEL
LIN {X 0,Y 521.154,Z 660.363,A -85,B 0,C 180,E1 25026.665,E2 25026.665} C_VEL
LIN {X 0,Y 520.916,Z 670.71,A -85,B 0,C 180,E1 25025.617,E2 25025.617} C_VEL
LIN {X 0,Y 520.695,Z 680.217,A -85,B 0,C 180,E1 25024.405,E2 25024.405} C_VEL
LIN {X 0,Y 520.499,Z 688.873,A -85,B 0,C 180,E1 25022.973,E2 25022.973} C_VEL
LIN {X 0,Y 520.343,Z 695.398,A -85,B 0,C 180,E1 25021.541,E2 25021.541} C_VEL
LIN {X 0,Y 520.257,Z 700.497,A -85,B 0,C 180,E1 25020,E2 25020} C_VEL
LIN {X 0,Y 520.196,Z 704.001,A -85,B 0,C 180,E1 25018.347,E2 25018.347} C_VEL
LIN {X 0,Y 520.177,Z 705.679,A -85,B 0,C 180,E1 25016.584,E2 25016.584} C_VEL
LIN {X 0,Y 520.159,Z 705.322,A -85,B 0,C 180,E1 25014.816,E2 25014.816} C_VEL
LIN {X 0,Y 520.185,Z 703.114,A -85,B 0,C 180,E1 25013.155,E2 25013.155} C_VEL
LIN {X 0,Y 520.22,Z 699.341,A -85,B 0,C 180,E1 25011.6,E2 25011.6} C_VEL
LIN {X 0,Y 520.323,Z 693.714,A -85,B 0,C 180,E1 25010.04,E2 25010.04} C_VEL
LIN {X 0,Y 520.48,Z 685.878,A -85,B 0,C 180,E1 25008.475,E2 25008.475} C_VEL
LIN {X 0,Y 520.682,Z 676.962,A -85,B 0,C 180,E1 25007.129,E2 25007.129} C_VEL
LIN {X 0,Y 520.911,Z 667.063,A -85,B 0,C 180,E1 25005.955,E2 25005.955} C_VEL
LIN {X 0,Y 521.17,Z 655.494,A -85,B 0,C 180,E1 25004.875,E2 25004.875} C_VEL
LIN {X 0,Y 521.451,Z 641.973,A -85,B 0,C 180,E1 25003.908,E2 25003.908} C_VEL
LIN {X 0,Y 521.666,Z 628.127,A -85,B 0,C 180,E1 25003.177,E2 25003.177} C_VEL
LIN {X 0,Y 521.828,Z 613.6,A -85,B 0,C 180,E1 25002.64,E2 25002.64} C_VEL
LIN {X 0,Y 521.922,Z 598.743,A -85,B 0,C 180,E1 25002.304,E2 25002.304} C_VEL
LIN {X 0,Y 522.213,Z 490.297,A -85,B 0,C 180,E1 25000.764,E2 25000.764} C_VEL
LIN {X 0,Y 522.929,Z 445.342,A -85,B 0,C 180,E1 24997.398,E2 24997.398} C_VEL
LIN {X 0,Y 523.166,Z 432.941,A -85,B 0,C 180,E1 24996.467,E2 24996.467} C_VEL
LIN {X 0,Y 522.326,Z 426.761,A -85,B 0,C 180,E1 24995.96,E2 24995.96} C_VEL
LIN {X 0,Y 516.631,Z 410.945,A -85,B 0,C 180,E1 24994.524,E2 24994.524} C_VEL
LIN {X 0,Y 516.017,Z 405.568,A -85,B 0,C 180,E1 24994.091,E2 24994.091} C_VEL
LIN {X 0,Y 516.747,Z 358.642,A -85,B 0,C 180,E1 24990.562,E2 24990.562} C_VEL
LIN {X 0,Y 517.289,Z 317.152,A -85,B 0,C 180,E1 24987.431,E2 24987.431} C_VEL
LIN {X 0,Y 517.785,Z 265.379,A -85,B 0,C 180,E1 24983.541,E2 24983.541} C_VEL
LIN {X 0,Y 512.645,Z 248.872,A -85,B 0,C 180,E1 24981.996,E2 24981.996} C_VEL
LIN {X 0,Y 512.648,Z 248.877,A -85,B 0,C 180,E1 24978.46,E2 24978.46} C_VEL
LIN {X 0,Y 512.614,Z 248.885,A -85,B 0,C 180,E1 24974.918,E2 24974.918} C_VEL
LIN {X 0,Y 512.649,Z 248.903,A -85,B 0,C 180,E1 24974.286,E2 24974.286} C_VEL
LIN {X 0,Y 513.955,Z 252.366,A -85,B 0,C 180,E1 24973.639,E2 24973.639} C_VEL
LIN {X 0,Y 515.029,Z 254.566,A -85,B 0,C 180,E1 24973.198,E2 24973.198} C_VEL
LIN {X 0,Y 519.153,Z 263.565,A -85,B 0,C 180,E1 24971.479,E2 24971.479} C_VEL
LIN {X 0,Y 524.873,Z 276.499,A -85,B 0,C 180,E1 24969.165,E2 24969.165} C_VEL
LIN {X 0,Y 525.58,Z 279.359,A -85,B 0,C 180,E1 24968.74,E2 24968.74} C_VEL
LIN {X 0,Y 523.027,Z 309.308,A -85,B 0,C 180,E1 24965.638,E2 24965.638} C_VEL
LIN {X 0,Y 524.973,Z 319.198,A -85,B 0,C 180,E1 24965.326,E2 24965.326} C_VEL
LIN {X 0,Y 521.816,Z 551.854,A -85,B 0,C 180,E1 24961.732,E2 24961.732} C_VEL
LIN {X 0,Y 521.362,Z 573.229,A -85,B 0,C 180,E1 24961.302,E2 24961.302} C_VEL
LIN {X 0,Y 520.667,Z 592.517,A -85,B 0,C 180,E1 24960.714,E2 24960.714} C_VEL
LIN {X 0,Y 519.888,Z 611.816,A -85,B 0,C 180,E1 24959.939,E2 24959.939} C_VEL
LIN {X 0,Y 518.903,Z 630.303,A -85,B 0,C 180,E1 24958.978,E2 24958.978} C_VEL
LIN {X 0,Y 518.006,Z 646.411,A -85,B 0,C 180,E1 24957.972,E2 24957.972} C_VEL
LIN {X 0,Y 516.91,Z 664.785,A -85,B 0,C 180,E1 24956.602,E2 24956.602} C_VEL
LIN {X 0,Y 515.946,Z 680.089,A -85,B 0,C 180,E1 24955.236,E2 24955.236} C_VEL
LIN {X 0,Y 515.077,Z 694.42,A -85,B 0,C 180,E1 24953.759,E2 24953.759} C_VEL
LIN {X 0,Y 514.171,Z 709.513,A -85,B 0,C 180,E1 24951.923,E2 24951.923} C_VEL
LIN {X 0,Y 513.492,Z 721.668,A -85,B 0,C 180,E1 24950.191,E2 24950.191} C_VEL
LIN {X 0,Y 512.917,Z 733.778,A -85,B 0,C 180,E1 24948.174,E2 24948.174} C_VEL
LIN {X 0,Y 512.498,Z 743.57,A -85,B 0,C 180,E1 24946.2,E2 24946.2} C_VEL
LIN {X 0,Y 512.227,Z 751.796,A -85,B 0,C 180,E1 24944.238,E2 24944.238} C_VEL
LIN {X 0,Y 512.045,Z 759.495,A -85,B 0,C 180,E1 24941.946,E2 24941.946} C_VEL
LIN {X 0,Y 511.962,Z 764.747,A -85,B 0,C 180,E1 24939.896,E2 24939.896} C_VEL
LIN {X 0,Y 511.928,Z 768.857,A -85,B 0,C 180,E1 24937.745,E2 24937.745} C_VEL
LIN {X 0,Y 511.904,Z 771.514,A -85,B 0,C 180,E1 24935.38,E2 24935.38} C_VEL
LIN {X 0,Y 511.904,Z 772.4,A -85,B 0,C 180,E1 24933.359,E2 24933.359} C_VEL
LIN {X 0,Y 511.909,Z 771.951,A -85,B 0,C 180,E1 24931.119,E2 24931.119} C_VEL
LIN {X 0,Y 511.915,Z 769.81,A -85,B 0,C 180,E1 24928.881,E2 24928.881} C_VEL
LIN {X 0,Y 511.939,Z 766.542,A -85,B 0,C 180,E1 24926.865,E2 24926.865} C_VEL
LIN {X 0,Y 512.011,Z 761.377,A -85,B 0,C 180,E1 24924.621,E2 24924.621} C_VEL
LIN {X 0,Y 512.163,Z 754.313,A -85,B 0,C 180,E1 24922.371,E2 24922.371} C_VEL
LIN {X 0,Y 512.39,Z 746.876,A -85,B 0,C 180,E1 24920.452,E2 24920.452} C_VEL
LIN {X 0,Y 512.808,Z 736.102,A -85,B 0,C 180,E1 24918.179,E2 24918.179} C_VEL
LIN {X 0,Y 513.287,Z 725.748,A -85,B 0,C 180,E1 24916.367,E2 24916.367} C_VEL
LIN {X 0,Y 513.994,Z 712.865,A -85,B 0,C 180,E1 24914.428,E2 24914.428} C_VEL
LIN {X 0,Y 514.795,Z 698.73,A -85,B 0,C 180,E1 24912.649,E2 24912.649} C_VEL
LIN {X 0,Y 515.665,Z 684.714,A -85,B 0,C 180,E1 24911.125,E2 24911.125} C_VEL
LIN {X 0,Y 516.769,Z 667.053,A -85,B 0,C 180,E1 24909.5,E2 24909.5} C_VEL
LIN {X 0,Y 517.652,Z 652.285,A -85,B 0,C 180,E1 24908.351,E2 24908.351} C_VEL
LIN {X 0,Y 518.62,Z 635.914,A -85,B 0,C 180,E1 24907.26,E2 24907.26} C_VEL
LIN {X 0,Y 519.662,Z 615.858,A -85,B 0,C 180,E1 24906.168,E2 24906.168} C_VEL
LIN {X 0,Y 520.439,Z 598.659,A -85,B 0,C 180,E1 24905.422,E2 24905.422} C_VEL
LIN {X 0,Y 521.184,Z 578.627,A -85,B 0,C 180,E1 24904.751,E2 24904.751} C_VEL
LIN {X 0,Y 521.681,Z 558.346,A -85,B 0,C 180,E1 24904.292,E2 24904.292} C_VEL
LIN {X 0,Y 525.028,Z 317.955,A -85,B 0,C 180,E1 24900.566,E2 24900.566} C_VEL
LIN {X 0,Y 524.646,Z 313.571,A -85,B 0,C 180,E1 24900.465,E2 24900.465} C_VEL
LIN {X 0,Y 523.507,Z 307.2,A -85,B 0,C 180,E1 24900.257,E2 24900.257} C_VEL
LIN {X 0,Y 525.58,Z 277.803,A -85,B 0,C 180,E1 24897.685,E2 24897.685} C_VEL
LIN {X 0,Y 521.804,Z 268.768,A -85,B 0,C 180,E1 24896.374,E2 24896.374} C_VEL
LIN {X 0,Y 515.968,Z 256.502,A -85,B 0,C 180,E1 24894.454,E2 24894.454} C_VEL
LIN {X 0,Y 514.068,Z 252.559,A -85,B 0,C 180,E1 24893.821,E2 24893.821} C_VEL
LIN {X 0,Y 512.649,Z 249.03,A -85,B 0,C 180,E1 24893.284,E2 24893.284} C_VEL
LIN {X 0,Y 512.637,Z 248.884,A -85,B 0,C 180,E1 24889.869,E2 24889.869} C_VEL
LIN {X 0,Y 512.649,Z 248.879,A -85,B 0,C 180,E1 24886.335,E2 24886.335} C_VEL
LIN {X 0,Y 512.625,Z 248.882,A -85,B 0,C 180,E1 24882.9,E2 24882.9} C_VEL
LIN {X 0,Y 512.628,Z 248.881,A -85,B 0,C 180,E1 24879.484,E2 24879.484} C_VEL
LIN {X 0,Y 512.646,Z 248.87,A -85,B 0,C 180,E1 24876.088,E2 24876.088} C_VEL
LIN {X 0,Y 512.649,Z 248.881,A -85,B 0,C 180,E1 24872.569,E2 24872.569} C_VEL
LIN {X 0,Y 512.666,Z 249.061,A -85,B 0,C 180,E1 24869.535,E2 24869.535} C_VEL
LIN {X 0,Y 518.015,Z 266.742,A -85,B 0,C 180,E1 24867.784,E2 24867.784} C_VEL
LIN {X 0,Y 517.59,Z 310.267,A -85,B 0,C 180,E1 24864.245,E2 24864.245} C_VEL
LIN {X 0,Y 517.024,Z 350.588,A -85,B 0,C 180,E1 24860.964,E2 24860.964} C_VEL
LIN {X 0,Y 516.265,Z 392.787,A -85,B 0,C 180,E1 24857.528,E2 24857.528} C_VEL
LIN {X 0,Y 515.445,Z 435.712,A -85,B 0,C 180,E1 24854.033,E2 24854.033} C_VEL
LIN {X 0,Y 515.397,Z 442.256,A -85,B 0,C 180,E1 24853.53,E2 24853.53} C_VEL
LIN {X 0,Y 515.777,Z 449.725,A -85,B 0,C 180,E1 24853.404,E2 24853.404} C_VEL
LIN {X 0,Y 514.902,Z 584.607,A -85,B 0,C 180,E1 24851.417,E2 24851.417} C_VEL
LIN {X 0,Y 514.744,Z 601.452,A -85,B 0,C 180,E1 24850.951,E2 24850.951} C_VEL
LIN {X 0,Y 514.469,Z 616.981,A -85,B 0,C 180,E1 24850.3,E2 24850.3} C_VEL
LIN {X 0,Y 514.15,Z 631.893,A -85,B 0,C 180,E1 24849.458,E2 24849.458} C_VEL
LIN {X 0,Y 513.767,Z 645.57,A -85,B 0,C 180,E1 24848.45,E2 24848.45} C_VEL
LIN {X 0,Y 513.401,Z 658.291,A -85,B 0,C 180,E1 24847.273,E2 24847.273} C_VEL
LIN {X 0,Y 513.038,Z 669.808,A -85,B 0,C 180,E1 24845.929,E2 24845.929} C_VEL
LIN {X 0,Y 512.74,Z 679.817,A -85,B 0,C 180,E1 24844.474,E2 24844.474} C_VEL
LIN {X 0,Y 512.5,Z 688.816,A -85,B 0,C 180,E1 24842.796,E2 24842.796} C_VEL
LIN {X 0,Y 512.368,Z 695.259,A -85,B 0,C 180,E1 24841.23,E2 24841.23} C_VEL
LIN {X 0,Y 512.262,Z 700.644,A -85,B 0,C 180,E1 24839.441,E2 24839.441} C_VEL
LIN {X 0,Y 512.228,Z 703.998,A -85,B 0,C 180,E1 24837.763,E2 24837.763} C_VEL
LIN {X 0,Y 512.204,Z 705.927,A -85,B 0,C 180,E1 24835.859,E2 24835.859} C_VEL
LIN {X 0,Y 512.223,Z 706.005,A -85,B 0,C 180,E1 24834.062,E2 24834.062} C_VEL
LIN {X 0,Y 512.261,Z 704.231,A -85,B 0,C 180,E1 24832.148,E2 24832.148} C_VEL
LIN {X 0,Y 512.333,Z 700.681,A -85,B 0,C 180,E1 24830.338,E2 24830.338} C_VEL
LIN {X 0,Y 512.455,Z 695.618,A -85,B 0,C 180,E1 24828.635,E2 24828.635} C_VEL
LIN {X 0,Y 512.615,Z 688.524,A -85,B 0,C 180,E1 24826.923,E2 24826.923} C_VEL
LIN {X 0,Y 512.857,Z 680.528,A -85,B 0,C 180,E1 24825.434,E2 24825.434} C_VEL
LIN {X 0,Y 513.138,Z 671.136,A -85,B 0,C 180,E1 24824.054,E2 24824.054} C_VEL
LIN {X 0,Y 513.501,Z 659.346,A -85,B 0,C 180,E1 24822.668,E2 24822.668} C_VEL
LIN {X 0,Y 513.841,Z 646.8,A -85,B 0,C 180,E1 24821.508,E2 24821.508} C_VEL
LIN {X 0,Y 514.167,Z 633.329,A -85,B 0,C 180,E1 24820.519,E2 24820.519} C_VEL
LIN {X 0,Y 514.427,Z 618.743,A -85,B 0,C 180,E1 24819.7,E2 24819.7} C_VEL
LIN {X 0,Y 514.64,Z 603.129,A -85,B 0,C 180,E1 24819.055,E2 24819.055} C_VEL
LIN {X 0,Y 514.732,Z 586.086,A -85,B 0,C 180,E1 24818.596,E2 24818.596} C_VEL
LIN {X 0,Y 515.586,Z 445.529,A -85,B 0,C 180,E1 24816.532,E2 24816.532} C_VEL
LIN {X 0,Y 516.105,Z 406.778,A -85,B 0,C 180,E1 24813.478,E2 24813.478} C_VEL
LIN {X 0,Y 516.329,Z 371.559,A -85,B 0,C 180,E1 24810.792,E2 24810.792} C_VEL
LIN {X 0,Y 516.196,Z 335.363,A -85,B 0,C 180,E1 24808.142,E2 24808.142} C_VEL
LIN {X 0,Y 515.92,Z 313.501,A -85,B 0,C 180,E1 24806.606,E2 24806.606} C_VEL
LIN {X 0,Y 515.457,Z 293.789,A -85,B 0,C 180,E1 24805.278,E2 24805.278} C_VEL
LIN {X 0,Y 515.162,Z 282.881,A -85,B 0,C 180,E1 24804.562,E2 24804.562} C_VEL
LIN {X 0,Y 516.327,Z 283.977,A -85,B 0,C 180,E1 24804.347,E2 24804.347} C_VEL
LIN {X 0,Y 518.433,Z 284.158,A -85,B 0,C 180,E1 24804.106,E2 24804.106} C_VEL
LIN {X 0,Y 520.898,Z 283.503,A -85,B 0,C 180,E1 24803.894,E2 24803.894} C_VEL
LIN {X 0,Y 524.585,Z 283.453,A -85,B 0,C 180,E1 24803.511,E2 24803.511} C_VEL
LIN {X 0,Y 526.915,Z 283.164,A -85,B 0,C 180,E1 24803.293,E2 24803.293} C_VEL
LIN {X 0,Y 529.331,Z 283.129,A -85,B 0,C 180,E1 24803.048,E2 24803.048} C_VEL
LIN {X 0,Y 530.07,Z 284.969,A -85,B 0,C 180,E1 24802.834,E2 24802.834} C_VEL
LIN {X 0,Y 528.314,Z 330.153,A -85,B 0,C 180,E1 24799.666,E2 24799.666} C_VEL
LIN {X 0,Y 529.474,Z 345.232,A -85,B 0,C 180,E1 24798.485,E2 24798.485} C_VEL
LIN {X 0,Y 532.254,Z 358.723,A -85,B 0,C 180,E1 24797.301,E2 24797.301} C_VEL
LIN {X 0,Y 536.237,Z 369.483,A -85,B 0,C 180,E1 24796.231,E2 24796.231} C_VEL
LIN {X 0,Y 541.699,Z 378.845,A -85,B 0,C 180,E1 24795.164,E2 24795.164} C_VEL
LIN {X 0,Y 548.665,Z 386.853,A -85,B 0,C 180,E1 24794.11,E2 24794.11} C_VEL
LIN {X 0,Y 557.154,Z 393.433,A -85,B 0,C 180,E1 24793.081,E2 24793.081} C_VEL
LIN {X 0,Y 566.453,Z 398.186,A -85,B 0,C 180,E1 24792.154,E2 24792.154} C_VEL
LIN {X 0,Y 571.404,Z 399.785,A -85,B 0,C 180,E1 24791.654,E2 24791.654} C_VEL
LIN {X 0,Y 575.271,Z 400.078,A -85,B 0,C 180,E1 24791.071,E2 24791.071} C_VEL
LIN {X 0,Y 577.704,Z 399.196,A -85,B 0,C 180,E1 24790.469,E2 24790.469} C_VEL
LIN {X 0,Y 578.762,Z 397.223,A -85,B 0,C 180,E1 24789.826,E2 24789.826} C_VEL
LIN {X 0,Y 578.267,Z 394.373,A -85,B 0,C 180,E1 24789.23,E2 24789.23} C_VEL
LIN {X 0,Y 576.227,Z 390.755,A -85,B 0,C 180,E1 24788.69,E2 24788.69} C_VEL
LIN {X 0,Y 570.059,Z 382.548,A -85,B 0,C 180,E1 24787.871,E2 24787.871} C_VEL
LIN {X 0,Y 567.994,Z 379.636,A -85,B 0,C 180,E1 24787.603,E2 24787.603} C_VEL
LIN {X 0,Y 564.259,Z 409.328,A -85,B 0,C 180,E1 24787.107,E2 24787.107} C_VEL
LIN {X 0,Y 561.649,Z 423.412,A -85,B 0,C 180,E1 24786.754,E2 24786.754} C_VEL
LIN {X 0,Y 560.493,Z 428.312,A -85,B 0,C 180,E1 24786.595,E2 24786.595} C_VEL
LIN {X 0,Y 558.164,Z 451.44,A -85,B 0,C 180,E1 24786.37,E2 24786.37} C_VEL
LIN {X 0,Y 554.061,Z 472.804,A -85,B 0,C 180,E1 24786.214,E2 24786.214} C_VEL
LIN {X 0,Y 548.472,Z 492.681,A -85,B 0,C 180,E1 24786.042,E2 24786.042} C_VEL
LIN {X 0,Y 543.228,Z 508.375,A -85,B 0,C 180,E1 24785.76,E2 24785.76} C_VEL
LIN {X 0,Y 539.565,Z 519.633,A -85,B 0,C 180,E1 24785.387,E2 24785.387} C_VEL
LIN {X 0,Y 538.69,Z 522.353,A -85,B 0,C 180,E1 24785.29,E2 24785.29} C_VEL
LIN {X 0,Y 534.011,Z 534.891,A -85,B 0,C 180,E1 24785.021,E2 24785.021} C_VEL
LIN {X 0,Y 530.505,Z 545.514,A -85,B 0,C 180,E1 24784.628,E2 24784.628} C_VEL
LIN {X 0,Y 528.93,Z 550.572,A -85,B 0,C 180,E1 24784.417,E2 24784.417} C_VEL
LIN {X 0,Y 525.846,Z 560.617,A -85,B 0,C 180,E1 24783.988,E2 24783.988} C_VEL
LIN {X 0,Y 524.959,Z 611.485,A -85,B 0,C 180,E1 24783.149,E2 24783.149} C_VEL
LIN {X 0,Y 524.153,Z 633.974,A -85,B 0,C 180,E1 24782.572,E2 24782.572} C_VEL
LIN {X 0,Y 523.217,Z 655.578,A -85,B 0,C 180,E1 24781.8,E2 24781.8} C_VEL
LIN {X 0,Y 522.021,Z 676.865,A -85,B 0,C 180,E1 24780.821,E2 24780.821} C_VEL
LIN {X 0,Y 520.789,Z 696.693,A -85,B 0,C 180,E1 24779.692,E2 24779.692} C_VEL
LIN {X 0,Y 519.423,Z 716.568,A -85,B 0,C 180,E1 24778.327,E2 24778.327} C_VEL
LIN {X 0,Y 518.04,Z 736.172,A -85,B 0,C 180,E1 24776.725,E2 24776.725} C_VEL
LIN {X 0,Y 516.753,Z 753.951,A -85,B 0,C 180,E1 24775.01,E2 24775.01} C_VEL
LIN {X 0,Y 515.559,Z 770.693,A -85,B 0,C 180,E1 24773.124,E2 24773.124} C_VEL
LIN {X 0,Y 514.514,Z 786.289,A -85,B 0,C 180,E1 24771.07,E2 24771.07} C_VEL
LIN {X 0,Y 513.643,Z 800.611,A -85,B 0,C 180,E1 24768.853,E2 24768.853} C_VEL
LIN {X 0,Y 512.969,Z 813.282,A -85,B 0,C 180,E1 24766.534,E2 24766.534} C_VEL
LIN {X 0,Y 512.488,Z 824.325,A -85,B 0,C 180,E1 24764.115,E2 24764.115} C_VEL
LIN {X 0,Y 512.197,Z 833.311,A -85,B 0,C 180,E1 24761.714,E2 24761.714} C_VEL
LIN {X 0,Y 512.036,Z 840.403,A -85,B 0,C 180,E1 24759.327,E2 24759.327} C_VEL
LIN {X 0,Y 511.95,Z 846.013,A -85,B 0,C 180,E1 24756.842,E2 24756.842} C_VEL
LIN {X 0,Y 511.92,Z 849.74,A -85,B 0,C 180,E1 24754.481,E2 24754.481} C_VEL
LIN {X 0,Y 511.91,Z 851.906,A -85,B 0,C 180,E1 24752.015,E2 24752.015} C_VEL
LIN {X 0,Y 511.897,Z 852.447,A -85,B 0,C 180,E1 24749.552,E2 24749.552} C_VEL
LIN {X 0,Y 511.912,Z 851.329,A -85,B 0,C 180,E1 24747.089,E2 24747.089} C_VEL
LIN {X 0,Y 511.926,Z 848.494,A -85,B 0,C 180,E1 24744.621,E2 24744.621} C_VEL
LIN {X 0,Y 511.975,Z 843.945,A -85,B 0,C 180,E1 24742.143,E2 24742.143} C_VEL
LIN {X 0,Y 512.084,Z 837.903,A -85,B 0,C 180,E1 24739.759,E2 24739.759} C_VEL
LIN {X 0,Y 512.292,Z 830.106,A -85,B 0,C 180,E1 24737.373,E2 24737.373} C_VEL
LIN {X 0,Y 512.649,Z 820.362,A -85,B 0,C 180,E1 24734.965,E2 24734.965} C_VEL
LIN {X 0,Y 513.18,Z 809.123,A -85,B 0,C 180,E1 24732.656,E2 24732.656} C_VEL
LIN {X 0,Y 513.946,Z 795.56,A -85,B 0,C 180,E1 24730.321,E2 24730.321} C_VEL
LIN {X 0,Y 514.909,Z 780.35,A -85,B 0,C 180,E1 24728.11,E2 24728.11} C_VEL
LIN {X 0,Y 516.056,Z 763.7,A -85,B 0,C 180,E1 24726.052,E2 24726.052} C_VEL
LIN {X 0,Y 517.373,Z 745.472,A -85,B 0,C 180,E1 24724.137,E2 24724.137} C_VEL
LIN {X 0,Y 518.711,Z 726.603,A -85,B 0,C 180,E1 24722.459,E2 24722.459} C_VEL
LIN {X 0,Y 520.129,Z 706.618,A -85,B 0,C 180,E1 24720.959,E2 24720.959} C_VEL
LIN {X 0,Y 521.429,Z 686.739,A -85,B 0,C 180,E1 24719.714,E2 24719.714} C_VEL
LIN {X 0,Y 522.658,Z 665.893,A -85,B 0,C 180,E1 24718.644,E2 24718.644} C_VEL
LIN {X 0,Y 523.756,Z 643.927,A -85,B 0,C 180,E1 24717.759,E2 24717.759} C_VEL
LIN {X 0,Y 524.611,Z 622.202,A -85,B 0,C 180,E1 24717.099,E2 24717.099} C_VEL
LIN {X 0,Y 525.241,Z 599.367,A -85,B 0,C 180,E1 24716.627,E2 24716.627} C_VEL
LIN {X 0,Y 525.697,Z 562.942,A -85,B 0,C 180,E1 24716.066,E2 24716.066} C_VEL
LIN {X 0,Y 528.445,Z 555.228,A -85,B 0,C 180,E1 24715.678,E2 24715.678} C_VEL
LIN {X 0,Y 530.231,Z 550.628,A -85,B 0,C 180,E1 24715.482,E2 24715.482} C_VEL
LIN {X 0,Y 533.731,Z 541.483,A -85,B 0,C 180,E1 24715.088,E2 24715.088} C_VEL
LIN {X 0,Y 538.777,Z 529.719,A -85,B 0,C 180,E1 24714.814,E2 24714.814} C_VEL
LIN {X 0,Y 539.958,Z 526.909,A -85,B 0,C 180,E1 24714.773,E2 24714.773} C_VEL
LIN {X 0,Y 543.322,Z 517.833,A -85,B 0,C 180,E1 24714.429,E2 24714.429} C_VEL
LIN {X 0,Y 548.294,Z 504.322,A -85,B 0,C 180,E1 24714.17,E2 24714.17} C_VEL
LIN {X 0,Y 553.679,Z 485.844,A -85,B 0,C 180,E1 24714.009,E2 24714.009} C_VEL
LIN {X 0,Y 557.057,Z 467.468,A -85,B 0,C 180,E1 24713.849,E2 24713.849} C_VEL
LIN {X 0,Y 560.754,Z 426.645,A -85,B 0,C 180,E1 24713.369,E2 24713.369} C_VEL
LIN {X 0,Y 563.187,Z 415.774,A -85,B 0,C 180,E1 24713.037,E2 24713.037} C_VEL
LIN {X 0,Y 564.203,Z 410.122,A -85,B 0,C 180,E1 24712.9,E2 24712.9} C_VEL
LIN {X 0,Y 570.29,Z 420.307,A -85,B 0,C 180,E1 24712.099,E2 24712.099} C_VEL
LIN {X 0,Y 573.541,Z 425.212,A -85,B 0,C 180,E1 24711.606,E2 24711.606} C_VEL
LIN {X 0,Y 575.074,Z 429.021,A -85,B 0,C 180,E1 24711.058,E2 24711.058} C_VEL
LIN {X 0,Y 575.1,Z 431.867,A -85,B 0,C 180,E1 24710.482,E2 24710.482} C_VEL
LIN {X 0,Y 573.616,Z 433.884,A -85,B 0,C 180,E1 24709.838,E2 24709.838} C_VEL
LIN {X 0,Y 571.128,Z 434.669,A -85,B 0,C 180,E1 24709.291,E2 24709.291} C_VEL
LIN {X 0,Y 567.625,Z 434.431,A -85,B 0,C 180,E1 24708.777,E2 24708.777} C_VEL
LIN {X 0,Y 562.689,Z 432.845,A -85,B 0,C 180,E1 24708.271,E2 24708.271} C_VEL
LIN {X 0,Y 552.68,Z 427.501,A -85,B 0,C 180,E1 24707.264,E2 24707.264} C_VEL
LIN {X 0,Y 544.304,Z 420.724,A -85,B 0,C 180,E1 24706.213,E2 24706.213} C_VEL
LIN {X 0,Y 537.544,Z 412.604,A -85,B 0,C 180,E1 24705.127,E2 24705.127} C_VEL
LIN {X 0,Y 532.236,Z 402.92,A -85,B 0,C 180,E1 24703.986,E2 24703.986} C_VEL
LIN {X 0,Y 528.653,Z 392.07,A -85,B 0,C 180,E1 24702.838,E2 24702.838} C_VEL
LIN {X 0,Y 526.399,Z 378.299,A -85,B 0,C 180,E1 24701.521,E2 24701.521} C_VEL
LIN {X 0,Y 525.992,Z 362.6,A -85,B 0,C 180,E1 24700.167,E2 24700.167} C_VEL
LIN {X 0,Y 528.734,Z 316.788,A -85,B 0,C 180,E1 24696.426,E2 24696.426} C_VEL
LIN {X 0,Y 530.726,Z 286.642,A -85,B 0,C 180,E1 24693.857,E2 24693.857} C_VEL
LIN {X 0,Y 523.076,Z 270.249,A -85,B 0,C 180,E1 24691.327,E2 24691.327} C_VEL
LIN {X 0,Y 518.643,Z 261.4,A -85,B 0,C 180,E1 24689.827,E2 24689.827} C_VEL
LIN {X 0,Y 516.478,Z 257.147,A -85,B 0,C 180,E1 24689.072,E2 24689.072} C_VEL
LIN {X 0,Y 514.769,Z 253.37,A -85,B 0,C 180,E1 24688.416,E2 24688.416} C_VEL
LIN {X 0,Y 513.471,Z 252.077,A -85,B 0,C 180,E1 24688.083,E2 24688.083} C_VEL
LIN {X 0,Y 514.984,Z 258.308,A -85,B 0,C 180,E1 24687.647,E2 24687.647} C_VEL
LIN {X 0,Y 515.619,Z 303.853,A -85,B 0,C 180,E1 24684.762,E2 24684.762} C_VEL
LIN {X 0,Y 516.042,Z 344.05,A -85,B 0,C 180,E1 24682.079,E2 24682.079} C_VEL
LIN {X 0,Y 516.013,Z 387.403,A -85,B 0,C 180,E1 24679.056,E2 24679.056} C_VEL
LIN {X 0,Y 515.578,Z 434.988,A -85,B 0,C 180,E1 24675.638,E2 24675.638} C_VEL
LIN {X 0,Y 514.943,Z 482.19,A -85,B 0,C 180,E1 24672.161,E2 24672.161} C_VEL
LIN {X 0,Y 514.635,Z 494.394,A -85,B 0,C 180,E1 24671.279,E2 24671.279} C_VEL
LIN {X 0,Y 514.054,Z 608.111,A -85,B 0,C 180,E1 24669.606,E2 24669.606} C_VEL
LIN {X 0,Y 513.962,Z 623.282,A -85,B 0,C 180,E1 24669.158,E2 24669.158} C_VEL
LIN {X 0,Y 513.822,Z 636.633,A -85,B 0,C 180,E1 24668.561,E2 24668.561} C_VEL
LIN {X 0,Y 513.592,Z 649.568,A -85,B 0,C 180,E1 24667.776,E2 24667.776} C_VEL
LIN {X 0,Y 513.35,Z 662.096,A -85,B 0,C 180,E1 24666.767,E2 24666.767} C_VEL
LIN {X 0,Y 513.072,Z 673.35,A -85,B 0,C 180,E1 24665.591,E2 24665.591} C_VEL
LIN {X 0,Y 512.845,Z 682.58,A -85,B 0,C 180,E1 24664.36,E2 24664.36} C_VEL
LIN {X 0,Y 512.652,Z 690.473,A -85,B 0,C 180,E1 24663.018,E2 24663.018} C_VEL
LIN {X 0,Y 512.475,Z 697.378,A -85,B 0,C 180,E1 24661.453,E2 24661.453} C_VEL
LIN {X 0,Y 512.379,Z 702.268,A -85,B 0,C 180,E1 24659.888,E2 24659.888} C_VEL
LIN {X 0,Y 512.311,Z 705.425,A -85,B 0,C 180,E1 24658.322,E2 24658.322} C_VEL
LIN {X 0,Y 512.287,Z 707.029,A -85,B 0,C 180,E1 24656.531,E2 24656.531} C_VEL
LIN {X 0,Y 512.27,Z 706.583,A -85,B 0,C 180,E1 24654.736,E2 24654.736} C_VEL
LIN {X 0,Y 512.3,Z 704.06,A -85,B 0,C 180,E1 24652.937,E2 24652.937} C_VEL
LIN {X 0,Y 512.355,Z 699.679,A -85,B 0,C 180,E1 24651.244,E2 24651.244} C_VEL
LIN {X 0,Y 512.473,Z 693.596,A -85,B 0,C 180,E1 24649.659,E2 24649.659} C_VEL
LIN {X 0,Y 512.633,Z 686.468,A -85,B 0,C 180,E1 24648.273,E2 24648.273} C_VEL
LIN {X 0,Y 512.857,Z 677.526,A -85,B 0,C 180,E1 24646.929,E2 24646.929} C_VEL
LIN {X 0,Y 513.118,Z 666.766,A -85,B 0,C 180,E1 24645.672,E2 24645.672} C_VEL
LIN {X 0,Y 513.374,Z 655.508,A -85,B 0,C 180,E1 24644.64,E2 24644.64} C_VEL
LIN {X 0,Y 513.657,Z 642.604,A -85,B 0,C 180,E1 24643.721,E2 24643.721} C_VEL
LIN {X 0,Y 513.881,Z 628.481,A -85,B 0,C 180,E1 24642.974,E2 24642.974} C_VEL
LIN {X 0,Y 514.046,Z 613.163,A -85,B 0,C 180,E1 24642.419,E2 24642.419} C_VEL
LIN {X 0,Y 514.121,Z 597.645,A -85,B 0,C 180,E1 24642.091,E2 24642.091} C_VEL
LIN {X 0,Y 514.517,Z 491.252,A -85,B 0,C 180,E1 24640.547,E2 24640.547} C_VEL
LIN {X 0,Y 515.273,Z 446.322,A -85,B 0,C 180,E1 24637.164,E2 24637.164} C_VEL
LIN {X 0,Y 516.017,Z 405.568,A -85,B 0,C 180,E1 24634.091,E2 24634.091} C_VEL
LIN {X 0,Y 515.18,Z 399.343,A -85,B 0,C 180,E1 24633.584,E2 24633.584} C_VEL
LIN {X 0,Y 509.345,Z 382.702,A -85,B 0,C 180,E1 24632.047,E2 24632.047} C_VEL
LIN {X 0,Y 508.897,Z 378.152,A -85,B 0,C 180,E1 24631.687,E2 24631.687} C_VEL
LIN {X 0,Y 509.57,Z 334.625,A -85,B 0,C 180,E1 24628.385,E2 24628.385} C_VEL
LIN {X 0,Y 509.978,Z 295.609,A -85,B 0,C 180,E1 24625.432,E2 24625.432} C_VEL
LIN {X 0,Y 510.127,Z 267.257,A -85,B 0,C 180,E1 24623.288,E2 24623.288} C_VEL
LIN {X 0,Y 504.712,Z 249.863,A -85,B 0,C 180,E1 24621.606,E2 24621.606} C_VEL
LIN {X 0,Y 504.705,Z 249.866,A -85,B 0,C 180,E1 24618.115,E2 24618.115} C_VEL
LIN {X 0,Y 504.71,Z 250.078,A -85,B 0,C 180,E1 24615.354,E2 24615.354} C_VEL
LIN {X 0,Y 506.112,Z 253.532,A -85,B 0,C 180,E1 24614.666,E2 24614.666} C_VEL
LIN {X 0,Y 507.09,Z 255.395,A -85,B 0,C 180,E1 24614.268,E2 24614.268} C_VEL
LIN {X 0,Y 510.979,Z 263.61,A -85,B 0,C 180,E1 24612.613,E2 24612.613} C_VEL
LIN {X 0,Y 517.411,Z 278.2,A -85,B 0,C 180,E1 24609.898,E2 24609.898} C_VEL
LIN {X 0,Y 519.172,Z 283.016,A -85,B 0,C 180,E1 24609.092,E2 24609.092} C_VEL
LIN {X 0,Y 516.617,Z 311.638,A -85,B 0,C 180,E1 24606.107,E2 24606.107} C_VEL
LIN {X 0,Y 518.414,Z 320.682,A -85,B 0,C 180,E1 24605.813,E2 24605.813} C_VEL
LIN {X 0,Y 515.799,Z 481.16,A -85,B 0,C 180,E1 24603.268,E2 24603.268} C_VEL
LIN {X 0,Y 514.485,Z 565.204,A -85,B 0,C 180,E1 24601.905,E2 24601.905} C_VEL
LIN {X 0,Y 513.833,Z 586.272,A -85,B 0,C 180,E1 24601.347,E2 24601.347} C_VEL
LIN {X 0,Y 512.988,Z 605.916,A -85,B 0,C 180,E1 24600.611,E2 24600.611} C_VEL
LIN {X 0,Y 511.987,Z 625.262,A -85,B 0,C 180,E1 24599.674,E2 24599.674} C_VEL
LIN {X 0,Y 510.877,Z 643.169,A -85,B 0,C 180,E1 24598.589,E2 24598.589} C_VEL
LIN {X 0,Y 509.863,Z 658.964,A -85,B 0,C 180,E1 24597.442,E2 24597.442} C_VEL
LIN {X 0,Y 508.61,Z 677.094,A -85,B 0,C 180,E1 24595.876,E2 24595.876} C_VEL
LIN {X 0,Y 507.63,Z 691.249,A -85,B 0,C 180,E1 24594.433,E2 24594.433} C_VEL
LIN {X 0,Y 506.701,Z 705.534,A -85,B 0,C 180,E1 24592.753,E2 24592.753} C_VEL
LIN {X 0,Y 505.833,Z 719.212,A -85,B 0,C 180,E1 24590.843,E2 24590.843} C_VEL
LIN {X 0,Y 505.218,Z 730.152,A -85,B 0,C 180,E1 24589.059,E2 24589.059} C_VEL
LIN {X 0,Y 504.677,Z 741.482,A -85,B 0,C 180,E1 24586.879,E2 24586.879} C_VEL
LIN {X 0,Y 504.321,Z 750.243,A -85,B 0,C 180,E1 24584.818,E2 24584.818} C_VEL
LIN {X 0,Y 504.102,Z 757.993,A -85,B 0,C 180,E1 24582.602,E2 24582.602} C_VEL
LIN {X 0,Y 503.977,Z 764.209,A -85,B 0,C 180,E1 24580.249,E2 24580.249} C_VEL
LIN {X 0,Y 503.934,Z 768.189,A -85,B 0,C 180,E1 24578.213,E2 24578.213} C_VEL
LIN {X 0,Y 503.915,Z 771.249,A -85,B 0,C 180,E1 24575.808,E2 24575.808} C_VEL
LIN {X 0,Y 503.903,Z 772.366,A -85,B 0,C 180,E1 24573.555,E2 24573.555} C_VEL
LIN {X 0,Y 503.902,Z 772.075,A -85,B 0,C 180,E1 24571.364,E2 24571.364} C_VEL
LIN {X 0,Y 503.918,Z 770.027,A -85,B 0,C 180,E1 24568.977,E2 24568.977} C_VEL
LIN {X 0,Y 503.941,Z 766.841,A -85,B 0,C 180,E1 24566.929,E2 24566.929} C_VEL
LIN {X 0,Y 504.012,Z 762.084,A -85,B 0,C 180,E1 24564.764,E2 24564.764} C_VEL
LIN {X 0,Y 504.18,Z 754.88,A -85,B 0,C 180,E1 24562.364,E2 24562.364} C_VEL
LIN {X 0,Y 504.423,Z 747.536,A -85,B 0,C 180,E1 24560.415,E2 24560.415} C_VEL
LIN {X 0,Y 504.855,Z 737.612,A -85,B 0,C 180,E1 24558.23,E2 24558.23} C_VEL
LIN {X 0,Y 505.401,Z 726.688,A -85,B 0,C 180,E1 24556.259,E2 24556.259} C_VEL
LIN {X 0,Y 506.046,Z 715.581,A -85,B 0,C 180,E1 24554.53,E2 24554.53} C_VEL
LIN {X 0,Y 507.003,Z 700.672,A -85,B 0,C 180,E1 24552.557,E2 24552.557} C_VEL
LIN {X 0,Y 507.909,Z 687.218,A -85,B 0,C 180,E1 24551.045,E2 24551.045} C_VEL
LIN {X 0,Y 508.894,Z 672.93,A -85,B 0,C 180,E1 24549.649,E2 24549.649} C_VEL
LIN {X 0,Y 510.104,Z 655.204,A -85,B 0,C 180,E1 24548.177,E2 24548.177} C_VEL
LIN {X 0,Y 511.125,Z 639.636,A -85,B 0,C 180,E1 24547.09,E2 24547.09} C_VEL
LIN {X 0,Y 512.181,Z 621.645,A -85,B 0,C 180,E1 24546.043,E2 24546.043} C_VEL
LIN {X 0,Y 513.166,Z 602.108,A -85,B 0,C 180,E1 24545.142,E2 24545.142} C_VEL
LIN {X 0,Y 513.965,Z 581.722,A -85,B 0,C 180,E1 24544.426,E2 24544.426} C_VEL
LIN {X 0,Y 514.577,Z 560.757,A -85,B 0,C 180,E1 24543.918,E2 24543.918} C_VEL
LIN {X 0,Y 518.217,Z 336.509,A -85,B 0,C 180,E1 24540.341,E2 24540.341} C_VEL
LIN {X 0,Y 518.32,Z 316.279,A -85,B 0,C 180,E1 24540.014,E2 24540.014} C_VEL
LIN {X 0,Y 517.101,Z 309.681,A -85,B 0,C 180,E1 24539.805,E2 24539.805} C_VEL
LIN {X 0,Y 519.138,Z 281.438,A -85,B 0,C 180,E1 24537.317,E2 24537.317} C_VEL
LIN {X 0,Y 512.689,Z 266.812,A -85,B 0,C 180,E1 24535.102,E2 24535.102} C_VEL
LIN {X 0,Y 506.2,Z 253.626,A -85,B 0,C 180,E1 24532.939,E2 24532.939} C_VEL
LIN {X 0,Y 504.773,Z 250.266,A -85,B 0,C 180,E1 24532.404,E2 24532.404} C_VEL
LIN {X 0,Y 504.713,Z 249.875,A -85,B 0,C 180,E1 24532.327,E2 24532.327} C_VEL
LIN {X 0,Y 504.694,Z 249.873,A -85,B 0,C 180,E1 24528.836,E2 24528.836} C_VEL
LIN {X 0,Y 504.688,Z 249.869,A -85,B 0,C 180,E1 24525.336,E2 24525.336} C_VEL
LIN {X 0,Y 504.693,Z 249.867,A -85,B 0,C 180,E1 24521.886,E2 24521.886} C_VEL
LIN {X 0,Y 504.71,Z 249.868,A -85,B 0,C 180,E1 24518.467,E2 24518.467} C_VEL
LIN {X 0,Y 504.702,Z 249.871,A -85,B 0,C 180,E1 24514.898,E2 24514.898} C_VEL
LIN {X 0,Y 504.702,Z 249.871,A -85,B 0,C 180,E1 24511.367,E2 24511.367} C_VEL
LIN {X 0,Y 504.721,Z 249.935,A -85,B 0,C 180,E1 24509.931,E2 24509.931} C_VEL
LIN {X 0,Y 510.578,Z 268.789,A -85,B 0,C 180,E1 24508.034,E2 24508.034} C_VEL
LIN {X 0,Y 510.11,Z 312.857,A -85,B 0,C 180,E1 24504.43,E2 24504.43} C_VEL
LIN {X 0,Y 509.482,Z 353.428,A -85,B 0,C 180,E1 24501.108,E2 24501.108} C_VEL
LIN {X 0,Y 508.671,Z 394.909,A -85,B 0,C 180,E1 24497.709,E2 24497.709} C_VEL
LIN {X 0,Y 507.812,Z 437.933,A -85,B 0,C 180,E1 24494.19,E2 24494.19} C_VEL
LIN {X 0,Y 507.802,Z 443.405,A -85,B 0,C 180,E1 24493.782,E2 24493.782} C_VEL
LIN {X 0,Y 508.131,Z 451.035,A -85,B 0,C 180,E1 24493.653,E2 24493.653} C_VEL
LIN {X 0,Y 507.154,Z 585.745,A -85,B 0,C 180,E1 24491.623,E2 24491.623} C_VEL
LIN {X 0,Y 506.997,Z 602.608,A -85,B 0,C 180,E1 24491.149,E2 24491.149} C_VEL
LIN {X 0,Y 506.728,Z 617.575,A -85,B 0,C 180,E1 24490.517,E2 24490.517} C_VEL
LIN {X 0,Y 506.395,Z 632.656,A -85,B 0,C 180,E1 24489.662,E2 24489.662} C_VEL
LIN {X 0,Y 505.994,Z 646.458,A -85,B 0,C 180,E1 24488.638,E2 24488.638} C_VEL
LIN {X 0,Y 505.607,Z 659.297,A -85,B 0,C 180,E1 24487.441,E2 24487.441} C_VEL
LIN {X 0,Y 505.209,Z 671.323,A -85,B 0,C 180,E1 24486.021,E2 24486.021} C_VEL
LIN {X 0,Y 504.89,Z 681.299,A -85,B 0,C 180,E1 24484.544,E2 24484.544} C_VEL
LIN {X 0,Y 504.637,Z 690.302,A -85,B 0,C 180,E1 24482.84,E2 24482.84} C_VEL
LIN {X 0,Y 504.479,Z 697.101,A -85,B 0,C 180,E1 24481.136,E2 24481.136} C_VEL
LIN {X 0,Y 504.382,Z 702.382,A -85,B 0,C 180,E1 24479.319,E2 24479.319} C_VEL
LIN {X 0,Y 504.333,Z 705.883,A -85,B 0,C 180,E1 24477.387,E2 24477.387} C_VEL
LIN {X 0,Y 504.321,Z 707.414,A -85,B 0,C 180,E1 24475.566,E2 24475.566} C_VEL
LIN {X 0,Y 504.353,Z 707.166,A -85,B 0,C 180,E1 24473.626,E2 24473.626} C_VEL
LIN {X 0,Y 504.391,Z 705.126,A -85,B 0,C 180,E1 24471.795,E2 24471.795} C_VEL
LIN {X 0,Y 504.506,Z 701.289,A -85,B 0,C 180,E1 24469.956,E2 24469.956} C_VEL
LIN {X 0,Y 504.631,Z 695.647,A -85,B 0,C 180,E1 24468.182,E2 24468.182} C_VEL
LIN {X 0,Y 504.849,Z 688.312,A -85,B 0,C 180,E1 24466.485,E2 24466.485} C_VEL
LIN {X 0,Y 505.133,Z 679.022,A -85,B 0,C 180,E1 24464.854,E2 24464.854} C_VEL
LIN {X 0,Y 505.464,Z 668.866,A -85,B 0,C 180,E1 24463.451,E2 24463.451} C_VEL
LIN {X 0,Y 505.849,Z 656.635,A -85,B 0,C 180,E1 24462.11,E2 24462.11} C_VEL
LIN {X 0,Y 506.166,Z 644.309,A -85,B 0,C 180,E1 24461.038,E2 24461.038} C_VEL
LIN {X 0,Y 506.516,Z 629.562,A -85,B 0,C 180,E1 24460.032,E2 24460.032} C_VEL
LIN {X 0,Y 506.755,Z 614.529,A -85,B 0,C 180,E1 24459.267,E2 24459.267} C_VEL
LIN {X 0,Y 506.915,Z 598.601,A -85,B 0,C 180,E1 24458.686,E2 24458.686} C_VEL
LIN {X 0,Y 506.948,Z 581.088,A -85,B 0,C 180,E1 24458.299,E2 24458.299} C_VEL
LIN {X 0,Y 507.845,Z 450.843,A -85,B 0,C 180,E1 24456.369,E2 24456.369} C_VEL
LIN {X 0,Y 507.932,Z 447.245,A -85,B 0,C 180,E1 24456.293,E2 24456.293} C_VEL
LIN {X 0,Y 508.519,Z 413.295,A -85,B 0,C 180,E1 24453.618,E2 24453.618} C_VEL
LIN {X 0,Y 508.801,Z 375.284,A -85,B 0,C 180,E1 24450.705,E2 24450.705} C_VEL
LIN {X 0,Y 508.632,Z 334.237,A -85,B 0,C 180,E1 24447.703,E2 24447.703} C_VEL
LIN {X 0,Y 508.293,Z 311.316,A -85,B 0,C 180,E1 24446.111,E2 24446.111} C_VEL
LIN {X 0,Y 507.814,Z 290.82,A -85,B 0,C 180,E1 24444.733,E2 24444.733} C_VEL
LIN {X 0,Y 509.31,Z 291.98,A -85,B 0,C 180,E1 24444.473,E2 24444.473} C_VEL
LIN {X 0,Y 511.521,Z 291.903,A -85,B 0,C 180,E1 24444.236,E2 24444.236} C_VEL
LIN {X 0,Y 513.274,Z 291.201,A -85,B 0,C 180,E1 24444.102,E2 24444.102} C_VEL
LIN {X 0,Y 516.945,Z 291.167,A -85,B 0,C 180,E1 24443.712,E2 24443.712} C_VEL
LIN {X 0,Y 519.318,Z 290.764,A -85,B 0,C 180,E1 24443.493,E2 24443.493} C_VEL
LIN {X 0,Y 523.545,Z 290.366,A -85,B 0,C 180,E1 24443.086,E2 24443.086} C_VEL
LIN {X 0,Y 521.763,Z 333.207,A -85,B 0,C 180,E1 24440.043,E2 24440.043} C_VEL
LIN {X 0,Y 522.939,Z 348.837,A -85,B 0,C 180,E1 24438.801,E2 24438.801} C_VEL
LIN {X 0,Y 525.667,Z 362.345,A -85,B 0,C 180,E1 24437.602,E2 24437.602} C_VEL
LIN {X 0,Y 529.794,Z 373.752,A -85,B 0,C 180,E1 24436.461,E2 24436.461} C_VEL
LIN {X 0,Y 535.173,Z 383.277,A -85,B 0,C 180,E1 24435.374,E2 24435.374} C_VEL
LIN {X 0,Y 542.621,Z 392.141,A -85,B 0,C 180,E1 24434.21,E2 24434.21} C_VEL
LIN {X 0,Y 551.023,Z 398.924,A -85,B 0,C 180,E1 24433.16,E2 24433.16} C_VEL
LIN {X 0,Y 560.94,Z 404.31,A -85,B 0,C 180,E1 24432.14,E2 24432.14} C_VEL
LIN {X 0,Y 567.59,Z 406.713,A -85,B 0,C 180,E1 24431.525,E2 24431.525} C_VEL
LIN {X 0,Y 571.785,Z 407.307,A -85,B 0,C 180,E1 24430.977,E2 24430.977} C_VEL
LIN {X 0,Y 574.761,Z 406.677,A -85,B 0,C 180,E1 24430.364,E2 24430.364} C_VEL
LIN {X 0,Y 576.224,Z 405.119,A -85,B 0,C 180,E1 24429.764,E2 24429.764} C_VEL
LIN {X 0,Y 576.278,Z 402.55,A -85,B 0,C 180,E1 24429.145,E2 24429.145} C_VEL
LIN {X 0,Y 574.796,Z 399.23,A -85,B 0,C 180,E1 24428.581,E2 24428.581} C_VEL
LIN {X 0,Y 571.752,Z 395.197,A -85,B 0,C 180,E1 24428.089,E2 24428.089} C_VEL
LIN {X 0,Y 571.231,Z 394.759,A -85,B 0,C 180,E1 24428.022,E2 24428.022} C_VEL
LIN {X 0,Y 567.827,Z 417.145,A -85,B 0,C 180,E1 24427.62,E2 24427.62} C_VEL
LIN {X 0,Y 564.995,Z 429.064,A -85,B 0,C 180,E1 24427.293,E2 24427.293} C_VEL
LIN {X 0,Y 561.131,Z 449.627,A -85,B 0,C 180,E1 24427.161,E2 24427.161} C_VEL
LIN {X 0,Y 555.367,Z 470.176,A -85,B 0,C 180,E1 24427.058,E2 24427.058} C_VEL
LIN {X 0,Y 547.927,Z 490.184,A -85,B 0,C 180,E1 24426.896,E2 24426.896} C_VEL
LIN {X 0,Y 540.946,Z 507.056,A -85,B 0,C 180,E1 24426.589,E2 24426.589} C_VEL
LIN {X 0,Y 536.484,Z 518.882,A -85,B 0,C 180,E1 24426.214,E2 24426.214} C_VEL
LIN {X 0,Y 535.11,Z 522.926,A -85,B 0,C 180,E1 24426.057,E2 24426.057} C_VEL
LIN {X 0,Y 529.283,Z 536.136,A -85,B 0,C 180,E1 24425.713,E2 24425.713} C_VEL
LIN {X 0,Y 525.457,Z 547.003,A -85,B 0,C 180,E1 24425.283,E2 24425.283} C_VEL
LIN {X 0,Y 520.894,Z 560.863,A -85,B 0,C 180,E1 24424.69,E2 24424.69} C_VEL
LIN {X 0,Y 518.986,Z 568.535,A -85,B 0,C 180,E1 24424.34,E2 24424.34} C_VEL
LIN {X 0,Y 518.3,Z 610.238,A -85,B 0,C 180,E1 24423.66,E2 24423.66} C_VEL
LIN {X 0,Y 517.46,Z 632.226,A -85,B 0,C 180,E1 24423.104,E2 24423.104} C_VEL
LIN {X 0,Y 516.442,Z 654.058,A -85,B 0,C 180,E1 24422.333,E2 24422.333} C_VEL
LIN {X 0,Y 515.216,Z 674.659,A -85,B 0,C 180,E1 24421.398,E2 24421.398} C_VEL
LIN {X 0,Y 513.822,Z 695.29,A -85,B 0,C 180,E1 24420.233,E2 24420.233} C_VEL
LIN {X 0,Y 512.348,Z 715.109,A -85,B 0,C 180,E1 24418.872,E2 24418.872} C_VEL
LIN {X 0,Y 510.817,Z 734.812,A -85,B 0,C 180,E1 24417.26,E2 24417.26} C_VEL
LIN {X 0,Y 509.379,Z 752.833,A -85,B 0,C 180,E1 24415.522,E2 24415.522} C_VEL
LIN {X 0,Y 508.014,Z 770.218,A -85,B 0,C 180,E1 24413.55,E2 24413.55} C_VEL
LIN {X 0,Y 506.807,Z 786.467,A -85,B 0,C 180,E1 24411.38,E2 24411.38} C_VEL
LIN {X 0,Y 505.84,Z 800.809,A -85,B 0,C 180,E1 24409.122,E2 24409.122} C_VEL
LIN {X 0,Y 505.105,Z 813.285,A -85,B 0,C 180,E1 24406.799,E2 24406.799} C_VEL
LIN {X 0,Y 504.555,Z 824.506,A -85,B 0,C 180,E1 24404.297,E2 24404.297} C_VEL
LIN {X 0,Y 504.221,Z 833.7,A -85,B 0,C 180,E1 24401.785,E2 24401.785} C_VEL
LIN {X 0,Y 504.04,Z 841,A -85,B 0,C 180,E1 24399.246,E2 24399.246} C_VEL
LIN {X 0,Y 503.952,Z 846.224,A -85,B 0,C 180,E1 24396.837,E2 24396.837} C_VEL
LIN {X 0,Y 503.919,Z 849.874,A -85,B 0,C 180,E1 24394.438,E2 24394.438} C_VEL
LIN {X 0,Y 503.907,Z 851.975,A -85,B 0,C 180,E1 24391.933,E2 24391.933} C_VEL
LIN {X 0,Y 503.897,Z 852.431,A -85,B 0,C 180,E1 24389.431,E2 24389.431} C_VEL
LIN {X 0,Y 503.915,Z 851.232,A -85,B 0,C 180,E1 24386.929,E2 24386.929} C_VEL
LIN {X 0,Y 503.93,Z 848.338,A -85,B 0,C 180,E1 24384.421,E2 24384.421} C_VEL
LIN {X 0,Y 503.989,Z 843.628,A -85,B 0,C 180,E1 24381.873,E2 24381.873} C_VEL
LIN {X 0,Y 504.119,Z 837.263,A -85,B 0,C 180,E1 24379.371,E2 24379.371} C_VEL
LIN {X 0,Y 504.367,Z 829.268,A -85,B 0,C 180,E1 24376.938,E2 24376.938} C_VEL
LIN {X 0,Y 504.763,Z 819.846,A -85,B 0,C 180,E1 24374.607,E2 24374.607} C_VEL
LIN {X 0,Y 505.369,Z 808.489,A -85,B 0,C 180,E1 24372.261,E2 24372.261} C_VEL
LIN {X 0,Y 506.181,Z 795.629,A -85,B 0,C 180,E1 24370.018,E2 24370.018} C_VEL
LIN {X 0,Y 507.253,Z 780.353,A -85,B 0,C 180,E1 24367.762,E2 24367.762} C_VEL
LIN {X 0,Y 508.523,Z 763.704,A -85,B 0,C 180,E1 24365.674,E2 24365.674} C_VEL
LIN {X 0,Y 509.957,Z 745.739,A -85,B 0,C 180,E1 24363.76,E2 24363.76} C_VEL
LIN {X 0,Y 511.395,Z 727.342,A -85,B 0,C 180,E1 24362.095,E2 24362.095} C_VEL
LIN {X 0,Y 512.927,Z 707.5,A -85,B 0,C 180,E1 24360.578,E2 24360.578} C_VEL
LIN {X 0,Y 514.346,Z 687.751,A -85,B 0,C 180,E1 24359.317,E2 24359.317} C_VEL
LIN {X 0,Y 515.681,Z 667.177,A -85,B 0,C 180,E1 24358.236,E2 24358.236} C_VEL
LIN {X 0,Y 516.888,Z 645.368,A -85,B 0,C 180,E1 24357.332,E2 24357.332} C_VEL
LIN {X 0,Y 517.822,Z 623.941,A -85,B 0,C 180,E1 24356.661,E2 24356.661} C_VEL
LIN {X 0,Y 518.516,Z 601.474,A -85,B 0,C 180,E1 24356.175,E2 24356.175} C_VEL
LIN {X 0,Y 519.088,Z 568.377,A -85,B 0,C 180,E1 24355.641,E2 24355.641} C_VEL
LIN {X 0,Y 523.258,Z 556.723,A -85,B 0,C 180,E1 24355.022,E2 24355.022} C_VEL
LIN {X 0,Y 525.756,Z 550.741,A -85,B 0,C 180,E1 24354.747,E2 24354.747} C_VEL
LIN {X 0,Y 529.86,Z 541.202,A -85,B 0,C 180,E1 24354.331,E2 24354.331} C_VEL
LIN {X 0,Y 536.022,Z 529.394,A -85,B 0,C 180,E1 24354.014,E2 24354.014} C_VEL
LIN {X 0,Y 537.366,Z 526.483,A -85,B 0,C 180,E1 24353.921,E2 24353.921} C_VEL
LIN {X 0,Y 542.001,Z 515.902,A -85,B 0,C 180,E1 24353.557,E2 24353.557} C_VEL
LIN {X 0,Y 548.144,Z 502.662,A -85,B 0,C 180,E1 24353.317,E2 24353.317} C_VEL
LIN {X 0,Y 555.192,Z 485.052,A -85,B 0,C 180,E1 24353.183,E2 24353.183} C_VEL
LIN {X 0,Y 560.37,Z 467.067,A -85,B 0,C 180,E1 24353.087,E2 24353.087} C_VEL
LIN {X 0,Y 563.494,Z 449.34,A -85,B 0,C 180,E1 24352.966,E2 24352.966} C_VEL
LIN {X 0,Y 565.449,Z 428.856,A -85,B 0,C 180,E1 24352.734,E2 24352.734} C_VEL
LIN {X 0,Y 566.472,Z 425.45,A -85,B 0,C 180,E1 24352.598,E2 24352.598} C_VEL
LIN {X 0,Y 570.71,Z 431.65,A -85,B 0,C 180,E1 24351.989,E2 24351.989} C_VEL
LIN {X 0,Y 572.377,Z 435.447,A -85,B 0,C 180,E1 24351.453,E2 24351.453} C_VEL
LIN {X 0,Y 572.522,Z 438.547,A -85,B 0,C 180,E1 24350.841,E2 24350.841} C_VEL
LIN {X 0,Y 571.164,Z 440.603,A -85,B 0,C 180,E1 24350.219,E2 24350.219} C_VEL
LIN {X 0,Y 568.418,Z 441.572,A -85,B 0,C 180,E1 24349.61,E2 24349.61} C_VEL
LIN {X 0,Y 564.443,Z 441.319,A -85,B 0,C 180,E1 24349.048,E2 24349.048} C_VEL
LIN {X 0,Y 559.102,Z 439.601,A -85,B 0,C 180,E1 24348.53,E2 24348.53} C_VEL
LIN {X 0,Y 548.968,Z 434.453,A -85,B 0,C 180,E1 24347.531,E2 24347.531} C_VEL
LIN {X 0,Y 540.405,Z 428.011,A -85,B 0,C 180,E1 24346.492,E2 24346.492} C_VEL
LIN {X 0,Y 533.378,Z 420.402,A -85,B 0,C 180,E1 24345.425,E2 24345.425} C_VEL
LIN {X 0,Y 527.832,Z 411.751,A -85,B 0,C 180,E1 24344.345,E2 24344.345} C_VEL
LIN {X 0,Y 523.371,Z 400.993,A -85,B 0,C 180,E1 24343.131,E2 24343.131} C_VEL
LIN {X 0,Y 520.427,Z 387.885,A -85,B 0,C 180,E1 24341.803,E2 24341.803} C_VEL
LIN {X 0,Y 519.253,Z 373.251,A -85,B 0,C 180,E1 24340.46,E2 24340.46} C_VEL
LIN {X 0,Y 520.467,Z 346.148,A -85,B 0,C 180,E1 24338.212,E2 24338.212} C_VEL
LIN {X 0,Y 523.188,Z 307.614,A -85,B 0,C 180,E1 24334.982,E2 24334.982} C_VEL
LIN {X 0,Y 524.36,Z 290.687,A -85,B 0,C 180,E1 24333.506,E2 24333.506} C_VEL
LIN {X 0,Y 517.171,Z 275.241,A -85,B 0,C 180,E1 24331.077,E2 24331.077} C_VEL
LIN {X 0,Y 511.315,Z 263.265,A -85,B 0,C 180,E1 24329.009,E2 24329.009} C_VEL
LIN {X 0,Y 509.476,Z 259.738,A -85,B 0,C 180,E1 24328.354,E2 24328.354} C_VEL
LIN {X 0,Y 507.787,Z 259.444,A -85,B 0,C 180,E1 24328.073,E2 24328.073} C_VEL
LIN {X 0,Y 507.3,Z 259.084,A -85,B 0,C 180,E1 24327.935,E2 24327.935} C_VEL
LIN {X 0,Y 508.027,Z 303.774,A -85,B 0,C 180,E1 24325.101,E2 24325.101} C_VEL
LIN {X 0,Y 508.45,Z 344.712,A -85,B 0,C 180,E1 24322.365,E2 24322.365} C_VEL
LIN {X 0,Y 508.412,Z 385.309,A -85,B 0,C 180,E1 24319.531,E2 24319.531} C_VEL
LIN {X 0,Y 508.006,Z 432.379,A -85,B 0,C 180,E1 24316.159,E2 24316.159} C_VEL
LIN {X 0,Y 507.395,Z 477.835,A -85,B 0,C 180,E1 24312.808,E2 24312.808} C_VEL
LIN {X 0,Y 506.896,Z 495.756,A -85,B 0,C 180,E1 24311.491,E2 24311.491} C_VEL
LIN {X 0,Y 506.25,Z 609.575,A -85,B 0,C 180,E1 24309.775,E2 24309.775} C_VEL
LIN {X 0,Y 506.169,Z 624.728,A -85,B 0,C 180,E1 24309.321,E2 24309.321} C_VEL
LIN {X 0,Y 506.029,Z 638.503,A -85,B 0,C 180,E1 24308.694,E2 24308.694} C_VEL
LIN {X 0,Y 505.793,Z 651.34,A -85,B 0,C 180,E1 24307.896,E2 24307.896} C_VEL
LIN {X 0,Y 505.539,Z 664.099,A -85,B 0,C 180,E1 24306.846,E2 24306.846} C_VEL
LIN {X 0,Y 505.255,Z 675.03,A -85,B 0,C 180,E1 24305.678,E2 24305.678} C_VEL
LIN {X 0,Y 505.013,Z 684.208,A -85,B 0,C 180,E1 24304.428,E2 24304.428} C_VEL
LIN {X 0,Y 504.805,Z 692.064,A -85,B 0,C 180,E1 24303.065,E2 24303.065} C_VEL
LIN {X 0,Y 504.615,Z 698.923,A -85,B 0,C 180,E1 24301.476,E2 24301.476} C_VEL
LIN {X 0,Y 504.504,Z 703.755,A -85,B 0,C 180,E1 24299.886,E2 24299.886} C_VEL
LIN {X 0,Y 504.426,Z 706.843,A -85,B 0,C 180,E1 24298.296,E2 24298.296} C_VEL
LIN {X 0,Y 504.399,Z 708.338,A -85,B 0,C 180,E1 24296.59,E2 24296.59} C_VEL
LIN {X 0,Y 504.376,Z 707.997,A -85,B 0,C 180,E1 24294.882,E2 24294.882} C_VEL
LIN {X 0,Y 504.399,Z 706.035,A -85,B 0,C 180,E1 24293.281,E2 24293.281} C_VEL
LIN {X 0,Y 504.451,Z 702.098,A -85,B 0,C 180,E1 24291.565,E2 24291.565} C_VEL
LIN {X 0,Y 504.568,Z 696.478,A -85,B 0,C 180,E1 24289.957,E2 24289.957} C_VEL
LIN {X 0,Y 504.737,Z 689.28,A -85,B 0,C 180,E1 24288.458,E2 24288.458} C_VEL
LIN {X 0,Y 504.958,Z 680.582,A -85,B 0,C 180,E1 24287.07,E2 24287.07} C_VEL
LIN {X 0,Y 505.234,Z 670.35,A -85,B 0,C 180,E1 24285.794,E2 24285.794} C_VEL
LIN {X 0,Y 505.531,Z 658.362,A -85,B 0,C 180,E1 24284.631,E2 24284.631} C_VEL
LIN {X 0,Y 505.826,Z 645.032,A -85,B 0,C 180,E1 24283.642,E2 24283.642} C_VEL
LIN {X 0,Y 506.063,Z 631.201,A -85,B 0,C 180,E1 24282.879,E2 24282.879} C_VEL
LIN {X 0,Y 506.227,Z 617.063,A -85,B 0,C 180,E1 24282.326,E2 24282.326} C_VEL
LIN {X 0,Y 506.312,Z 601.85,A -85,B 0,C 180,E1 24281.956,E2 24281.956} C_VEL
LIN {X 0,Y 506.829,Z 492.077,A -85,B 0,C 180,E1 24280.314,E2 24280.314} C_VEL
LIN {X 0,Y 507.638,Z 446.58,A -85,B 0,C 180,E1 24276.868,E2 24276.868} C_VEL
LIN {X 0,Y 508.508,Z 401.201,A -85,B 0,C 180,E1 24273.427,E2 24273.427} C_VEL
LIN {X 0,Y 508.897,Z 378.152,A -85,B 0,C 180,E1 24271.687,E2 24271.687} C_VEL
LIN {X 0,Y 508.168,Z 371.924,A -85,B 0,C 180,E1 24271.17,E2 24271.17} C_VEL
LIN {X 0,Y 502.459,Z 356.194,A -85,B 0,C 180,E1 24269.678,E2 24269.678} C_VEL
LIN {X 0,Y 501.852,Z 350.807,A -85,B 0,C 180,E1 24269.235,E2 24269.235} C_VEL
LIN {X 0,Y 502.459,Z 304.677,A -85,B 0,C 180,E1 24265.725,E2 24265.725} C_VEL
LIN {X 0,Y 502.765,Z 269.919,A -85,B 0,C 180,E1 24263.08,E2 24263.08} C_VEL
LIN {X 0,Y 496.755,Z 250.859,A -85,B 0,C 180,E1 24261.246,E2 24261.246} C_VEL
LIN {X 0,Y 496.773,Z 250.857,A -85,B 0,C 180,E1 24257.603,E2 24257.603} C_VEL
LIN {X 0,Y 496.736,Z 250.863,A -85,B 0,C 180,E1 24256.551,E2 24256.551} C_VEL
LIN {X 0,Y 498.055,Z 254.33,A -85,B 0,C 180,E1 24255.844,E2 24255.844} C_VEL
LIN {X 0,Y 499.123,Z 256.26,A -85,B 0,C 180,E1 24255.401,E2 24255.401} C_VEL
LIN {X 0,Y 501.583,Z 261.451,A -85,B 0,C 180,E1 24254.304,E2 24254.304} C_VEL
LIN {X 0,Y 505.173,Z 269.012,A -85,B 0,C 180,E1 24252.751,E2 24252.751} C_VEL
LIN {X 0,Y 511.551,Z 283.709,A -85,B 0,C 180,E1 24249.986,E2 24249.986} C_VEL
LIN {X 0,Y 512.757,Z 287.137,A -85,B 0,C 180,E1 24249.406,E2 24249.406} C_VEL
LIN {X 0,Y 510.213,Z 313.853,A -85,B 0,C 180,E1 24246.592,E2 24246.592} C_VEL
LIN {X 0,Y 511.893,Z 322.223,A -85,B 0,C 180,E1 24246.312,E2 24246.312} C_VEL
LIN {X 0,Y 509.579,Z 449.48,A -85,B 0,C 180,E1 24244.26,E2 24244.26} C_VEL
LIN {X 0,Y 507.36,Z 566.54,A -85,B 0,C 180,E1 24242.296,E2 24242.296} C_VEL
LIN {X 0,Y 506.665,Z 587.75,A -85,B 0,C 180,E1 24241.719,E2 24241.719} C_VEL
LIN {X 0,Y 505.733,Z 608.244,A -85,B 0,C 180,E1 24240.933,E2 24240.933} C_VEL
LIN {X 0,Y 504.707,Z 626.655,A -85,B 0,C 180,E1 24240.015,E2 24240.015} C_VEL
LIN {X 0,Y 503.532,Z 644.478,A -85,B 0,C 180,E1 24238.916,E2 24238.916} C_VEL
LIN {X 0,Y 502.284,Z 662.469,A -85,B 0,C 180,E1 24237.57,E2 24237.57} C_VEL
LIN {X 0,Y 500.987,Z 679.325,A -85,B 0,C 180,E1 24236.045,E2 24236.045} C_VEL
LIN {X 0,Y 499.913,Z 693.076,A -85,B 0,C 180,E1 24234.583,E2 24234.583} C_VEL
LIN {X 0,Y 498.763,Z 708.767,A -85,B 0,C 180,E1 24232.638,E2 24232.638} C_VEL
LIN {X 0,Y 497.966,Z 720.427,A -85,B 0,C 180,E1 24230.941,E2 24230.941} C_VEL
LIN {X 0,Y 497.299,Z 731.431,A -85,B 0,C 180,E1 24229.094,E2 24229.094} C_VEL
LIN {X 0,Y 496.708,Z 742.599,A -85,B 0,C 180,E1 24226.85,E2 24226.85} C_VEL
LIN {X 0,Y 496.36,Z 750.501,A -85,B 0,C 180,E1 24224.942,E2 24224.942} C_VEL
LIN {X 0,Y 496.118,Z 758.204,A -85,B 0,C 180,E1 24222.69,E2 24222.69} C_VEL
LIN {X 0,Y 495.983,Z 764.277,A -85,B 0,C 180,E1 24220.335,E2 24220.335} C_VEL
LIN {X 0,Y 495.935,Z 768.104,A -85,B 0,C 180,E1 24218.347,E2 24218.347} C_VEL
LIN {X 0,Y 495.919,Z 771.101,A -85,B 0,C 180,E1 24216.018,E2 24216.018} C_VEL
LIN {X 0,Y 495.905,Z 772.342,A -85,B 0,C 180,E1 24213.699,E2 24213.699} C_VEL
LIN {X 0,Y 495.9,Z 772.165,A -85,B 0,C 180,E1 24211.618,E2 24211.618} C_VEL
LIN {X 0,Y 495.914,Z 770.521,A -85,B 0,C 180,E1 24209.307,E2 24209.307} C_VEL
LIN {X 0,Y 495.944,Z 767.14,A -85,B 0,C 180,E1 24206.995,E2 24206.995} C_VEL
LIN {X 0,Y 496.009,Z 762.742,A -85,B 0,C 180,E1 24204.911,E2 24204.911} C_VEL
LIN {X 0,Y 496.175,Z 756.249,A -85,B 0,C 180,E1 24202.59,E2 24202.59} C_VEL
LIN {X 0,Y 496.433,Z 748.666,A -85,B 0,C 180,E1 24200.494,E2 24200.494} C_VEL
LIN {X 0,Y 496.829,Z 740.051,A -85,B 0,C 180,E1 24198.508,E2 24198.508} C_VEL
LIN {X 0,Y 497.471,Z 728.423,A -85,B 0,C 180,E1 24196.281,E2 24196.281} C_VEL
LIN {X 0,Y 498.152,Z 717.478,A -85,B 0,C 180,E1 24194.517,E2 24194.517} C_VEL
LIN {X 0,Y 498.98,Z 705.707,A -85,B 0,C 180,E1 24192.869,E2 24192.869} C_VEL
LIN {X 0,Y 500.201,Z 689.495,A -85,B 0,C 180,E1 24190.924,E2 24190.924} C_VEL
LIN {X 0,Y 501.37,Z 674.429,A -85,B 0,C 180,E1 24189.391,E2 24189.391} C_VEL
LIN {X 0,Y 502.661,Z 657.165,A -85,B 0,C 180,E1 24187.917,E2 24187.917} C_VEL
LIN {X 0,Y 503.892,Z 639.793,A -85,B 0,C 180,E1 24186.68,E2 24186.68} C_VEL
LIN {X 0,Y 505.01,Z 621.389,A -85,B 0,C 180,E1 24185.61,E2 24185.61} C_VEL
LIN {X 0,Y 506.013,Z 602.436,A -85,B 0,C 180,E1 24184.735,E2 24184.735} C_VEL
LIN {X 0,Y 506.831,Z 582.391,A -85,B 0,C 180,E1 24184.026,E2 24184.026} C_VEL
LIN {X 0,Y 507.467,Z 562.038,A -85,B 0,C 180,E1 24183.523,E2 24183.523} C_VEL
LIN {X 0,Y 511.381,Z 356.022,A -85,B 0,C 180,E1 24180.128,E2 24180.128} C_VEL
LIN {X 0,Y 511.806,Z 317.672,A -85,B 0,C 180,E1 24179.511,E2 24179.511} C_VEL
LIN {X 0,Y 510.748,Z 311.713,A -85,B 0,C 180,E1 24179.306,E2 24179.306} C_VEL
LIN {X 0,Y 512.778,Z 285.392,A -85,B 0,C 180,E1 24176.978,E2 24176.978} C_VEL
LIN {X 0,Y 506.056,Z 270.663,A -85,B 0,C 180,E1 24174.687,E2 24174.687} C_VEL
LIN {X 0,Y 500.267,Z 258.692,A -85,B 0,C 180,E1 24172.7,E2 24172.7} C_VEL
LIN {X 0,Y 498.401,Z 254.793,A -85,B 0,C 180,E1 24172.038,E2 24172.038} C_VEL
LIN {X 0,Y 496.833,Z 251.356,A -85,B 0,C 180,E1 24171.457,E2 24171.457} C_VEL
LIN {X 0,Y 496.753,Z 250.866,A -85,B 0,C 180,E1 24171.35,E2 24171.35} C_VEL
LIN {X 0,Y 496.757,Z 250.86,A -85,B 0,C 180,E1 24167.913,E2 24167.913} C_VEL
LIN {X 0,Y 496.775,Z 250.858,A -85,B 0,C 180,E1 24164.397,E2 24164.397} C_VEL
LIN {X 0,Y 496.764,Z 250.843,A -85,B 0,C 180,E1 24160.703,E2 24160.703} C_VEL
LIN {X 0,Y 496.754,Z 250.844,A -85,B 0,C 180,E1 24157.146,E2 24157.146} C_VEL
LIN {X 0,Y 496.756,Z 250.86,A -85,B 0,C 180,E1 24153.609,E2 24153.609} C_VEL
LIN {X 0,Y 496.783,Z 250.948,A -85,B 0,C 180,E1 24150.329,E2 24150.329} C_VEL
LIN {X 0,Y 503.183,Z 271.657,A -85,B 0,C 180,E1 24148.225,E2 24148.225} C_VEL
LIN {X 0,Y 502.627,Z 315.428,A -85,B 0,C 180,E1 24144.619,E2 24144.619} C_VEL
LIN {X 0,Y 501.967,Z 354.795,A -85,B 0,C 180,E1 24141.378,E2 24141.378} C_VEL
LIN {X 0,Y 501.115,Z 396.387,A -85,B 0,C 180,E1 24137.955,E2 24137.955} C_VEL
LIN {X 0,Y 500.209,Z 438.722,A -85,B 0,C 180,E1 24134.47,E2 24134.47} C_VEL
LIN {X 0,Y 500.19,Z 444.338,A -85,B 0,C 180,E1 24134.046,E2 24134.046} C_VEL
LIN {X 0,Y 500.49,Z 452.035,A -85,B 0,C 180,E1 24133.912,E2 24133.912} C_VEL
LIN {X 0,Y 499.409,Z 587.031,A -85,B 0,C 180,E1 24131.831,E2 24131.831} C_VEL
LIN {X 0,Y 499.255,Z 603.891,A -85,B 0,C 180,E1 24131.348,E2 24131.348} C_VEL
LIN {X 0,Y 498.966,Z 619.304,A -85,B 0,C 180,E1 24130.682,E2 24130.682} C_VEL
LIN {X 0,Y 498.623,Z 634.274,A -85,B 0,C 180,E1 24129.814,E2 24129.814} C_VEL
LIN {X 0,Y 498.188,Z 648.701,A -85,B 0,C 180,E1 24128.716,E2 24128.716} C_VEL
LIN {X 0,Y 497.775,Z 661.317,A -85,B 0,C 180,E1 24127.503,E2 24127.503} C_VEL
LIN {X 0,Y 497.379,Z 672.825,A -85,B 0,C 180,E1 24126.117,E2 24126.117} C_VEL
LIN {X 0,Y 497.039,Z 682.773,A -85,B 0,C 180,E1 24124.616,E2 24124.616} C_VEL
LIN {X 0,Y 496.783,Z 691.235,A -85,B 0,C 180,E1 24123,E2 24123} C_VEL
LIN {X 0,Y 496.625,Z 697.78,A -85,B 0,C 180,E1 24121.385,E2 24121.385} C_VEL
LIN {X 0,Y 496.501,Z 703.257,A -85,B 0,C 180,E1 24119.539,E2 24119.539} C_VEL
LIN {X 0,Y 496.457,Z 706.667,A -85,B 0,C 180,E1 24117.807,E2 24117.807} C_VEL
LIN {X 0,Y 496.435,Z 708.651,A -85,B 0,C 180,E1 24115.842,E2 24115.842} C_VEL
LIN {X 0,Y 496.465,Z 708.725,A -85,B 0,C 180,E1 24113.989,E2 24113.989} C_VEL
LIN {X 0,Y 496.516,Z 707.084,A -85,B 0,C 180,E1 24112.13,E2 24112.13} C_VEL
LIN {X 0,Y 496.6,Z 703.869,A -85,B 0,C 180,E1 24110.38,E2 24110.38} C_VEL
LIN {X 0,Y 496.765,Z 698.534,A -85,B 0,C 180,E1 24108.507,E2 24108.507} C_VEL
LIN {X 0,Y 496.941,Z 691.964,A -85,B 0,C 180,E1 24106.859,E2 24106.859} C_VEL
LIN {X 0,Y 497.24,Z 683.368,A -85,B 0,C 180,E1 24105.205,E2 24105.205} C_VEL
LIN {X 0,Y 497.588,Z 672.993,A -85,B 0,C 180,E1 24103.662,E2 24103.662} C_VEL
LIN {X 0,Y 497.958,Z 661.94,A -85,B 0,C 180,E1 24102.351,E2 24102.351} C_VEL
LIN {X 0,Y 498.33,Z 649.194,A -85,B 0,C 180,E1 24101.154,E2 24101.154} C_VEL
LIN {X 0,Y 498.65,Z 636.329,A -85,B 0,C 180,E1 24100.193,E2 24100.193} C_VEL
LIN {X 0,Y 498.914,Z 621.579,A -85,B 0,C 180,E1 24099.347,E2 24099.347} C_VEL
LIN {X 0,Y 499.111,Z 606.101,A -85,B 0,C 180,E1 24098.695,E2 24098.695} C_VEL
LIN {X 0,Y 499.172,Z 588.931,A -85,B 0,C 180,E1 24098.223,E2 24098.223} C_VEL
LIN {X 0,Y 500.216,Z 449.47,A -85,B 0,C 180,E1 24096.077,E2 24096.077} C_VEL
LIN {X 0,Y 500.658,Z 442.476,A -85,B 0,C 180,E1 24095.534,E2 24095.534} C_VEL
LIN {X 0,Y 501.143,Z 402.832,A -85,B 0,C 180,E1 24092.428,E2 24092.428} C_VEL
LIN {X 0,Y 501.301,Z 364.997,A -85,B 0,C 180,E1 24089.562,E2 24089.562} C_VEL
LIN {X 0,Y 501.027,Z 327.377,A -85,B 0,C 180,E1 24086.853,E2 24086.853} C_VEL
LIN {X 0,Y 500.56,Z 300.915,A -85,B 0,C 180,E1 24085.021,E2 24085.021} C_VEL
LIN {X 0,Y 500.553,Z 298.985,A -85,B 0,C 180,E1 24084.881,E2 24084.881} C_VEL
LIN {X 0,Y 502.282,Z 300.016,A -85,B 0,C 180,E1 24084.601,E2 24084.601} C_VEL
LIN {X 0,Y 504.585,Z 299.711,A -85,B 0,C 180,E1 24084.369,E2 24084.369} C_VEL
LIN {X 0,Y 506.306,Z 299.082,A -85,B 0,C 180,E1 24084.23,E2 24084.23} C_VEL
LIN {X 0,Y 510.027,Z 298.916,A -85,B 0,C 180,E1 24083.838,E2 24083.838} C_VEL
LIN {X 0,Y 512.423,Z 298.452,A -85,B 0,C 180,E1 24083.618,E2 24083.618} C_VEL
LIN {X 0,Y 516.899,Z 297.887,A -85,B 0,C 180,E1 24083.191,E2 24083.191} C_VEL
LIN {X 0,Y 515.225,Z 335.765,A -85,B 0,C 180,E1 24080.467,E2 24080.467} C_VEL
LIN {X 0,Y 516.316,Z 351.679,A -85,B 0,C 180,E1 24079.189,E2 24079.189} C_VEL
LIN {X 0,Y 518.924,Z 365.344,A -85,B 0,C 180,E1 24077.967,E2 24077.967} C_VEL
LIN {X 0,Y 522.907,Z 377.016,A -85,B 0,C 180,E1 24076.801,E2 24076.801} C_VEL
LIN {X 0,Y 528.659,Z 387.691,A -85,B 0,C 180,E1 24075.591,E2 24075.591} C_VEL
LIN {X 0,Y 536.2,Z 397.013,A -85,B 0,C 180,E1 24074.369,E2 24074.369} C_VEL
LIN {X 0,Y 544.906,Z 404.381,A -85,B 0,C 180,E1 24073.243,E2 24073.243} C_VEL
LIN {X 0,Y 554.706,Z 410.062,A -85,B 0,C 180,E1 24072.198,E2 24072.198} C_VEL
LIN {X 0,Y 565.12,Z 413.952,A -85,B 0,C 180,E1 24071.241,E2 24071.241} C_VEL
LIN {X 0,Y 568.942,Z 414.476,A -85,B 0,C 180,E1 24070.761,E2 24070.761} C_VEL
LIN {X 0,Y 572.102,Z 413.938,A -85,B 0,C 180,E1 24070.158,E2 24070.158} C_VEL
LIN {X 0,Y 573.674,Z 412.645,A -85,B 0,C 180,E1 24069.614,E2 24069.614} C_VEL
LIN {X 0,Y 574.085,Z 410.315,A -85,B 0,C 180,E1 24068.998,E2 24068.998} C_VEL
LIN {X 0,Y 573.269,Z 408.046,A -85,B 0,C 180,E1 24068.523,E2 24068.523} C_VEL
LIN {X 0,Y 568.866,Z 425.48,A -85,B 0,C 180,E1 24068.214,E2 24068.214} C_VEL
LIN {X 0,Y 566.735,Z 432.879,A -85,B 0,C 180,E1 24068.026,E2 24068.026} C_VEL
LIN {X 0,Y 560.738,Z 452.697,A -85,B 0,C 180,E1 24067.965,E2 24067.965} C_VEL
LIN {X 0,Y 552.803,Z 472.428,A -85,B 0,C 180,E1 24067.851,E2 24067.851} C_VEL
LIN {X 0,Y 543.736,Z 491.172,A -85,B 0,C 180,E1 24067.626,E2 24067.626} C_VEL
LIN {X 0,Y 535.955,Z 506.996,A -85,B 0,C 180,E1 24067.256,E2 24067.256} C_VEL
LIN {X 0,Y 530.796,Z 519.464,A -85,B 0,C 180,E1 24066.816,E2 24066.816} C_VEL
LIN {X 0,Y 529.622,Z 522.595,A -85,B 0,C 180,E1 24066.692,E2 24066.692} C_VEL
LIN {X 0,Y 523.118,Z 535.702,A -85,B 0,C 180,E1 24066.268,E2 24066.268} C_VEL
LIN {X 0,Y 518.918,Z 547.07,A -85,B 0,C 180,E1 24065.788,E2 24065.788} C_VEL
LIN {X 0,Y 514.07,Z 561.404,A -85,B 0,C 180,E1 24065.15,E2 24065.15} C_VEL
LIN {X 0,Y 512.28,Z 568.591,A -85,B 0,C 180,E1 24064.828,E2 24064.828} C_VEL
LIN {X 0,Y 511.609,Z 610.282,A -85,B 0,C 180,E1 24064.152,E2 24064.152} C_VEL
LIN {X 0,Y 510.774,Z 631.598,A -85,B 0,C 180,E1 24063.616,E2 24063.616} C_VEL
LIN {X 0,Y 509.666,Z 653.289,A -85,B 0,C 180,E1 24062.85,E2 24062.85} C_VEL
LIN {X 0,Y 508.4,Z 673.306,A -85,B 0,C 180,E1 24061.941,E2 24061.941} C_VEL
LIN {X 0,Y 506.899,Z 693.827,A -85,B 0,C 180,E1 24060.788,E2 24060.788} C_VEL
LIN {X 0,Y 505.366,Z 713.322,A -85,B 0,C 180,E1 24059.456,E2 24059.456} C_VEL
LIN {X 0,Y 503.751,Z 732.094,A -85,B 0,C 180,E1 24057.932,E2 24057.932} C_VEL
LIN {X 0,Y 502.103,Z 751.096,A -85,B 0,C 180,E1 24056.11,E2 24056.11} C_VEL
LIN {X 0,Y 500.63,Z 768.234,A -85,B 0,C 180,E1 24054.169,E2 24054.169} C_VEL
LIN {X 0,Y 499.346,Z 783.753,A -85,B 0,C 180,E1 24052.113,E2 24052.113} C_VEL
LIN {X 0,Y 498.275,Z 797.776,A -85,B 0,C 180,E1 24049.946,E2 24049.946} C_VEL
LIN {X 0,Y 497.422,Z 810.336,A -85,B 0,C 180,E1 24047.669,E2 24047.669} C_VEL
LIN {X 0,Y 496.791,Z 821.407,A -85,B 0,C 180,E1 24045.287,E2 24045.287} C_VEL
LIN {X 0,Y 496.361,Z 830.929,A -85,B 0,C 180,E1 24042.802,E2 24042.802} C_VEL
LIN {X 0,Y 496.101,Z 838.892,A -85,B 0,C 180,E1 24040.216,E2 24040.216} C_VEL
LIN {X 0,Y 495.977,Z 844.678,A -85,B 0,C 180,E1 24037.763,E2 24037.763} C_VEL
LIN {X 0,Y 495.927,Z 848.817,A -85,B 0,C 180,E1 24035.321,E2 24035.321} C_VEL
LIN {X 0,Y 495.911,Z 851.5,A -85,B 0,C 180,E1 24032.774,E2 24032.774} C_VEL
LIN {X 0,Y 495.904,Z 852.475,A -85,B 0,C 180,E1 24030.231,E2 24030.231} C_VEL
LIN {X 0,Y 495.91,Z 851.844,A -85,B 0,C 180,E1 24027.805,E2 24027.805} C_VEL
LIN {X 0,Y 495.923,Z 849.588,A -85,B 0,C 180,E1 24025.258,E2 24025.258} C_VEL
LIN {X 0,Y 495.965,Z 845.562,A -85,B 0,C 180,E1 24022.685,E2 24022.685} C_VEL
LIN {X 0,Y 496.07,Z 839.803,A -85,B 0,C 180,E1 24020.135,E2 24020.135} C_VEL
LIN {X 0,Y 496.297,Z 832.528,A -85,B 0,C 180,E1 24017.669,E2 24017.669} C_VEL
LIN {X 0,Y 496.673,Z 823.861,A -85,B 0,C 180,E1 24015.306,E2 24015.306} C_VEL
LIN {X 0,Y 497.284,Z 812.71,A -85,B 0,C 180,E1 24012.808,E2 24012.808} C_VEL
LIN {X 0,Y 498.124,Z 799.91,A -85,B 0,C 180,E1 24010.414,E2 24010.414} C_VEL
LIN {X 0,Y 499.214,Z 785.448,A -85,B 0,C 180,E1 24008.128,E2 24008.128} C_VEL
LIN {X 0,Y 500.549,Z 769.234,A -85,B 0,C 180,E1 24005.952,E2 24005.952} C_VEL
LIN {X 0,Y 502.001,Z 752.271,A -85,B 0,C 180,E1 24004.012,E2 24004.012} C_VEL
LIN {X 0,Y 503.638,Z 733.45,A -85,B 0,C 180,E1 24002.19,E2 24002.19} C_VEL
LIN {X 0,Y 505.286,Z 714.194,A -85,B 0,C 180,E1 24000.61,E2 24000.61} C_VEL
LIN {X 0,Y 506.83,Z 694.815,A -85,B 0,C 180,E1 23999.273,E2 23999.273} C_VEL
LIN {X 0,Y 508.322,Z 674.529,A -85,B 0,C 180,E1 23998.12,E2 23998.12} C_VEL
LIN {X 0,Y 509.631,Z 653.975,A -85,B 0,C 180,E1 23997.178,E2 23997.178} C_VEL
LIN {X 0,Y 510.766,Z 631.845,A -85,B 0,C 180,E1 23996.392,E2 23996.392} C_VEL
LIN {X 0,Y 511.606,Z 610.459,A -85,B 0,C 180,E1 23995.852,E2 23995.852} C_VEL
LIN {X 0,Y 512.263,Z 569.548,A -85,B 0,C 180,E1 23995.188,E2 23995.188} C_VEL
LIN {X 0,Y 513.028,Z 566.404,A -85,B 0,C 180,E1 23995.041,E2 23995.041} C_VEL
LIN {X 0,Y 517.072,Z 555.76,A -85,B 0,C 180,E1 23994.473,E2 23994.473} C_VEL
LIN {X 0,Y 523.508,Z 541.493,A -85,B 0,C 180,E1 23993.781,E2 23993.781} C_VEL
LIN {X 0,Y 529.812,Z 530.778,A -85,B 0,C 180,E1 23993.39,E2 23993.39} C_VEL
LIN {X 0,Y 532.312,Z 526.55,A -85,B 0,C 180,E1 23993.255,E2 23993.255} C_VEL
LIN {X 0,Y 537.386,Z 516.265,A -85,B 0,C 180,E1 23992.86,E2 23992.86} C_VEL
LIN {X 0,Y 545.001,Z 502.817,A -85,B 0,C 180,E1 23992.542,E2 23992.542} C_VEL
LIN {X 0,Y 553.919,Z 486.048,A -85,B 0,C 180,E1 23992.367,E2 23992.367} C_VEL
LIN {X 0,Y 560.813,Z 469.766,A -85,B 0,C 180,E1 23992.289,E2 23992.289} C_VEL
LIN {X 0,Y 566.111,Z 452.499,A -85,B 0,C 180,E1 23992.234,E2 23992.234} C_VEL
LIN {X 0,Y 568.831,Z 439.773,A -85,B 0,C 180,E1 23992.16,E2 23992.16} C_VEL
LIN {X 0,Y 570.022,Z 443.401,A -85,B 0,C 180,E1 23991.583,E2 23991.583} C_VEL
LIN {X 0,Y 569.734,Z 445.945,A -85,B 0,C 180,E1 23991.027,E2 23991.027} C_VEL
LIN {X 0,Y 568.092,Z 447.743,A -85,B 0,C 180,E1 23990.421,E2 23990.421} C_VEL
LIN {X 0,Y 565.176,Z 448.523,A -85,B 0,C 180,E1 23989.84,E2 23989.84} C_VEL
LIN {X 0,Y 561.453,Z 448.231,A -85,B 0,C 180,E1 23989.344,E2 23989.344} C_VEL
LIN {X 0,Y 555.527,Z 446.352,A -85,B 0,C 180,E1 23988.792,E2 23988.792} C_VEL
LIN {X 0,Y 545.283,Z 441.369,A -85,B 0,C 180,E1 23987.799,E2 23987.799} C_VEL
LIN {X 0,Y 535.916,Z 434.678,A -85,B 0,C 180,E1 23986.687,E2 23986.687} C_VEL
LIN {X 0,Y 528.165,Z 426.691,A -85,B 0,C 180,E1 23985.536,E2 23985.536} C_VEL
LIN {X 0,Y 522.01,Z 417.508,A -85,B 0,C 180,E1 23984.356,E2 23984.356} C_VEL
LIN {X 0,Y 517.287,Z 406.702,A -85,B 0,C 180,E1 23983.1,E2 23983.1} C_VEL
LIN {X 0,Y 514.134,Z 393.949,A -85,B 0,C 180,E1 23981.764,E2 23981.764} C_VEL
LIN {X 0,Y 512.648,Z 379.101,A -85,B 0,C 180,E1 23980.355,E2 23980.355} C_VEL
LIN {X 0,Y 513.155,Z 359.444,A -85,B 0,C 180,E1 23978.671,E2 23978.671} C_VEL
LIN {X 0,Y 516.243,Z 318.689,A -85,B 0,C 180,E1 23975.251,E2 23975.251} C_VEL
LIN {X 0,Y 518.069,Z 294.926,A -85,B 0,C 180,E1 23973.171,E2 23973.171} C_VEL
LIN {X 0,Y 511.285,Z 280.214,A -85,B 0,C 180,E1 23970.821,E2 23970.821} C_VEL
LIN {X 0,Y 505.457,Z 268.347,A -85,B 0,C 180,E1 23968.73,E2 23968.73} C_VEL
LIN {X 0,Y 504.42,Z 266.807,A -85,B 0,C 180,E1 23968.406,E2 23968.406} C_VEL
LIN {X 0,Y 502.09,Z 267.694,A -85,B 0,C 180,E1 23968.161,E2 23968.161} C_VEL
LIN {X 0,Y 500.132,Z 267.348,A -85,B 0,C 180,E1 23967.827,E2 23967.827} C_VEL
LIN {X 0,Y 499.962,Z 267.32,A -85,B 0,C 180,E1 23967.773,E2 23967.773} C_VEL
LIN {X 0,Y 500.58,Z 311.797,A -85,B 0,C 180,E1 23964.926,E2 23964.926} C_VEL
LIN {X 0,Y 500.892,Z 351.839,A -85,B 0,C 180,E1 23962.222,E2 23962.222} C_VEL
LIN {X 0,Y 500.789,Z 394.836,A -85,B 0,C 180,E1 23959.198,E2 23959.198} C_VEL
LIN {X 0,Y 500.371,Z 438.306,A -85,B 0,C 180,E1 23956.066,E2 23956.066} C_VEL
LIN {X 0,Y 499.698,Z 485.193,A -85,B 0,C 180,E1 23952.597,E2 23952.597} C_VEL
LIN {X 0,Y 499.204,Z 496.904,A -85,B 0,C 180,E1 23951.729,E2 23951.729} C_VEL
LIN {X 0,Y 498.453,Z 611.525,A -85,B 0,C 180,E1 23949.941,E2 23949.941} C_VEL
LIN {X 0,Y 498.382,Z 626.801,A -85,B 0,C 180,E1 23949.468,E2 23949.468} C_VEL
LIN {X 0,Y 498.242,Z 640.398,A -85,B 0,C 180,E1 23948.83,E2 23948.83} C_VEL
LIN {X 0,Y 498.001,Z 653.137,A -85,B 0,C 180,E1 23948.021,E2 23948.021} C_VEL
LIN {X 0,Y 497.743,Z 665.57,A -85,B 0,C 180,E1 23946.98,E2 23946.98} C_VEL
LIN {X 0,Y 497.439,Z 676.853,A -85,B 0,C 180,E1 23945.752,E2 23945.752} C_VEL
LIN {X 0,Y 497.184,Z 685.845,A -85,B 0,C 180,E1 23944.498,E2 23944.498} C_VEL
LIN {X 0,Y 496.957,Z 693.654,A -85,B 0,C 180,E1 23943.114,E2 23943.114} C_VEL
LIN {X 0,Y 496.754,Z 700.469,A -85,B 0,C 180,E1 23941.499,E2 23941.499} C_VEL
LIN {X 0,Y 496.622,Z 705.524,A -85,B 0,C 180,E1 23939.769,E2 23939.769} C_VEL
LIN {X 0,Y 496.537,Z 708.55,A -85,B 0,C 180,E1 23938.038,E2 23938.038} C_VEL
LIN {X 0,Y 496.504,Z 709.704,A -85,B 0,C 180,E1 23936.42,E2 23936.42} C_VEL
LIN {X 0,Y 496.488,Z 709.177,A -85,B 0,C 180,E1 23934.684,E2 23934.684} C_VEL
LIN {X 0,Y 496.518,Z 706.777,A -85,B 0,C 180,E1 23932.944,E2 23932.944} C_VEL
LIN {X 0,Y 496.574,Z 702.779,A -85,B 0,C 180,E1 23931.314,E2 23931.314} C_VEL
LIN {X 0,Y 496.704,Z 697.381,A -85,B 0,C 180,E1 23929.796,E2 23929.796} C_VEL
LIN {X 0,Y 496.909,Z 689.391,A -85,B 0,C 180,E1 23928.156,E2 23928.156} C_VEL
LIN {X 0,Y 497.161,Z 680.306,A -85,B 0,C 180,E1 23926.745,E2 23926.745} C_VEL
LIN {X 0,Y 497.442,Z 670.124,A -85,B 0,C 180,E1 23925.508,E2 23925.508} C_VEL
LIN {X 0,Y 497.746,Z 658.375,A -85,B 0,C 180,E1 23924.384,E2 23924.384} C_VEL
LIN {X 0,Y 498.044,Z 645.551,A -85,B 0,C 180,E1 23923.436,E2 23923.436} C_VEL
LIN {X 0,Y 498.287,Z 631.497,A -85,B 0,C 180,E1 23922.663,E2 23922.663} C_VEL
LIN {X 0,Y 498.448,Z 616.93,A -85,B 0,C 180,E1 23922.104,E2 23922.104} C_VEL
LIN {X 0,Y 498.516,Z 601.958,A -85,B 0,C 180,E1 23921.751,E2 23921.751} C_VEL
LIN {X 0,Y 499.143,Z 493.1,A -85,B 0,C 180,E1 23920.09,E2 23920.09} C_VEL
LIN {X 0,Y 500.002,Z 447.537,A -85,B 0,C 180,E1 23916.618,E2 23916.618} C_VEL
LIN {X 0,Y 500.936,Z 401.734,A -85,B 0,C 180,E1 23913.122,E2 23913.122} C_VEL
LIN {X 0,Y 501.743,Z 356.084,A -85,B 0,C 180,E1 23909.641,E2 23909.641} C_VEL
LIN {X 0,Y 501.852,Z 350.807,A -85,B 0,C 180,E1 23909.235,E2 23909.235} C_VEL
LIN {X 0,Y 501.02,Z 344.548,A -85,B 0,C 180,E1 23908.718,E2 23908.718} C_VEL
LIN {X 0,Y 495.201,Z 327.867,A -85,B 0,C 180,E1 23907.137,E2 23907.137} C_VEL
LIN {X 0,Y 494.758,Z 323.358,A -85,B 0,C 180,E1 23906.764,E2 23906.764} C_VEL
LIN {X 0,Y 495.523,Z 272.932,A -85,B 0,C 180,E1 23902.892,E2 23902.892} C_VEL
LIN {X 0,Y 488.797,Z 251.851,A -85,B 0,C 180,E1 23900.85,E2 23900.85} C_VEL
LIN {X 0,Y 488.848,Z 251.953,A -85,B 0,C 180,E1 23897.767,E2 23897.767} C_VEL
LIN {X 0,Y 490.12,Z 255.32,A -85,B 0,C 180,E1 23897.049,E2 23897.049} C_VEL
LIN {X 0,Y 491.185,Z 257.057,A -85,B 0,C 180,E1 23896.612,E2 23896.612} C_VEL
LIN {X 0,Y 493.818,Z 262.755,A -85,B 0,C 180,E1 23895.364,E2 23895.364} C_VEL
LIN {X 0,Y 496.148,Z 267.54,A -85,B 0,C 180,E1 23894.322,E2 23894.322} C_VEL
LIN {X 0,Y 500.903,Z 277.818,A -85,B 0,C 180,E1 23892.22,E2 23892.22} C_VEL
LIN {X 0,Y 506.424,Z 290.939,A -85,B 0,C 180,E1 23889.769,E2 23889.769} C_VEL
LIN {X 0,Y 503.907,Z 316.296,A -85,B 0,C 180,E1 23887.081,E2 23887.081} C_VEL
LIN {X 0,Y 505.413,Z 323.831,A -85,B 0,C 180,E1 23886.823,E2 23886.823} C_VEL
LIN {X 0,Y 503.207,Z 435.613,A -85,B 0,C 180,E1 23884.994,E2 23884.994} C_VEL
LIN {X 0,Y 500.249,Z 568.035,A -85,B 0,C 180,E1 23882.695,E2 23882.695} C_VEL
LIN {X 0,Y 499.501,Z 589.306,A -85,B 0,C 180,E1 23882.096,E2 23882.096} C_VEL
LIN {X 0,Y 498.507,Z 609.573,A -85,B 0,C 180,E1 23881.298,E2 23881.298} C_VEL
LIN {X 0,Y 497.355,Z 628.965,A -85,B 0,C 180,E1 23880.305,E2 23880.305} C_VEL
LIN {X 0,Y 496.066,Z 647.455,A -85,B 0,C 180,E1 23879.128,E2 23879.128} C_VEL
LIN {X 0,Y 494.731,Z 665.113,A -85,B 0,C 180,E1 23877.759,E2 23877.759} C_VEL
LIN {X 0,Y 493.383,Z 681.646,A -85,B 0,C 180,E1 23876.218,E2 23876.218} C_VEL
LIN {X 0,Y 492.083,Z 697.287,A -85,B 0,C 180,E1 23874.488,E2 23874.488} C_VEL
LIN {X 0,Y 490.92,Z 711.291,A -85,B 0,C 180,E1 23872.64,E2 23872.64} C_VEL
LIN {X 0,Y 489.998,Z 723.203,A -85,B 0,C 180,E1 23870.797,E2 23870.797} C_VEL
LIN {X 0,Y 489.198,Z 735.413,A -85,B 0,C 180,E1 23868.593,E2 23868.593} C_VEL
LIN {X 0,Y 488.697,Z 744.477,A -85,B 0,C 180,E1 23866.645,E2 23866.645} C_VEL
LIN {X 0,Y 488.312,Z 753.193,A -85,B 0,C 180,E1 23864.416,E2 23864.416} C_VEL
LIN {X 0,Y 488.086,Z 760.038,A -85,B 0,C 180,E1 23862.181,E2 23862.181} C_VEL
LIN {X 0,Y 487.98,Z 764.934,A -85,B 0,C 180,E1 23860.149,E2 23860.149} C_VEL
LIN {X 0,Y 487.931,Z 769.158,A -85,B 0,C 180,E1 23857.773,E2 23857.773} C_VEL
LIN {X 0,Y 487.904,Z 771.56,A -85,B 0,C 180,E1 23855.409,E2 23855.409} C_VEL
LIN {X 0,Y 487.903,Z 772.386,A -85,B 0,C 180,E1 23853.407,E2 23853.407} C_VEL
LIN {X 0,Y 487.91,Z 771.975,A -85,B 0,C 180,E1 23851.057,E2 23851.057} C_VEL
LIN {X 0,Y 487.912,Z 769.84,A -85,B 0,C 180,E1 23848.708,E2 23848.708} C_VEL
LIN {X 0,Y 487.945,Z 766.796,A -85,B 0,C 180,E1 23846.711,E2 23846.711} C_VEL
LIN {X 0,Y 488.03,Z 762.301,A -85,B 0,C 180,E1 23844.592,E2 23844.592} C_VEL
LIN {X 0,Y 488.235,Z 755.21,A -85,B 0,C 180,E1 23842.114,E2 23842.114} C_VEL
LIN {X 0,Y 488.533,Z 747.92,A -85,B 0,C 180,E1 23840.101,E2 23840.101} C_VEL
LIN {X 0,Y 489.02,Z 738.652,A -85,B 0,C 180,E1 23837.962,E2 23837.962} C_VEL
LIN {X 0,Y 489.714,Z 727.319,A -85,B 0,C 180,E1 23835.818,E2 23835.818} C_VEL
LIN {X 0,Y 490.648,Z 714.872,A -85,B 0,C 180,E1 23833.788,E2 23833.788} C_VEL
LIN {X 0,Y 491.812,Z 700.439,A -85,B 0,C 180,E1 23831.816,E2 23831.816} C_VEL
LIN {X 0,Y 493.021,Z 686.025,A -85,B 0,C 180,E1 23830.142,E2 23830.142} C_VEL
LIN {X 0,Y 494.451,Z 668.836,A -85,B 0,C 180,E1 23828.466,E2 23828.466} C_VEL
LIN {X 0,Y 495.803,Z 651.323,A -85,B 0,C 180,E1 23827.058,E2 23827.058} C_VEL
LIN {X 0,Y 497.065,Z 633.22,A -85,B 0,C 180,E1 23825.856,E2 23825.856} C_VEL
LIN {X 0,Y 498.193,Z 615.214,A -85,B 0,C 180,E1 23824.882,E2 23824.882} C_VEL
LIN {X 0,Y 499.187,Z 595.574,A -85,B 0,C 180,E1 23824.039,E2 23824.039} C_VEL
LIN {X 0,Y 500.003,Z 576.149,A -85,B 0,C 180,E1 23823.417,E2 23823.417} C_VEL
LIN {X 0,Y 500.557,Z 555.734,A -85,B 0,C 180,E1 23822.968,E2 23822.968} C_VEL
LIN {X 0,Y 504.693,Z 366.777,A -85,B 0,C 180,E1 23819.771,E2 23819.771} C_VEL
LIN {X 0,Y 505.35,Z 319.216,A -85,B 0,C 180,E1 23818.998,E2 23818.998} C_VEL
LIN {X 0,Y 504.412,Z 313.931,A -85,B 0,C 180,E1 23818.811,E2 23818.811} C_VEL
LIN {X 0,Y 506.391,Z 289.454,A -85,B 0,C 180,E1 23816.638,E2 23816.638} C_VEL
LIN {X 0,Y 498.976,Z 273.046,A -85,B 0,C 180,E1 23814.047,E2 23814.047} C_VEL
LIN {X 0,Y 492.491,Z 259.905,A -85,B 0,C 180,E1 23811.785,E2 23811.785} C_VEL
LIN {X 0,Y 490.678,Z 256.077,A -85,B 0,C 180,E1 23811.116,E2 23811.116} C_VEL
LIN {X 0,Y 489.004,Z 252.761,A -85,B 0,C 180,E1 23810.513,E2 23810.513} C_VEL
LIN {X 0,Y 488.835,Z 251.852,A -85,B 0,C 180,E1 23810.345,E2 23810.345} C_VEL
LIN {X 0,Y 488.829,Z 251.845,A -85,B 0,C 180,E1 23806.734,E2 23806.734} C_VEL
LIN {X 0,Y 488.815,Z 251.847,A -85,B 0,C 180,E1 23803.094,E2 23803.094} C_VEL
LIN {X 0,Y 488.815,Z 251.843,A -85,B 0,C 180,E1 23799.543,E2 23799.543} C_VEL
LIN {X 0,Y 488.828,Z 251.833,A -85,B 0,C 180,E1 23796.092,E2 23796.092} C_VEL
LIN {X 0,Y 488.832,Z 251.848,A -85,B 0,C 180,E1 23792.544,E2 23792.544} C_VEL
LIN {X 0,Y 488.838,Z 252.029,A -85,B 0,C 180,E1 23790.726,E2 23790.726} C_VEL
LIN {X 0,Y 495.76,Z 274.26,A -85,B 0,C 180,E1 23788.437,E2 23788.437} C_VEL
LIN {X 0,Y 495.177,Z 317.028,A -85,B 0,C 180,E1 23784.898,E2 23784.898} C_VEL
LIN {X 0,Y 494.439,Z 357.705,A -85,B 0,C 180,E1 23781.53,E2 23781.53} C_VEL
LIN {X 0,Y 493.51,Z 399.622,A -85,B 0,C 180,E1 23778.059,E2 23778.059} C_VEL
LIN {X 0,Y 492.555,Z 442.361,A -85,B 0,C 180,E1 23774.519,E2 23774.519} C_VEL
LIN {X 0,Y 492.573,Z 445.243,A -85,B 0,C 180,E1 23774.315,E2 23774.315} C_VEL
LIN {X 0,Y 492.856,Z 453.065,A -85,B 0,C 180,E1 23774.177,E2 23774.177} C_VEL
LIN {X 0,Y 491.672,Z 588.268,A -85,B 0,C 180,E1 23772.046,E2 23772.046} C_VEL
LIN {X 0,Y 491.519,Z 604.994,A -85,B 0,C 180,E1 23771.559,E2 23771.559} C_VEL
LIN {X 0,Y 491.21,Z 621.023,A -85,B 0,C 180,E1 23770.853,E2 23770.853} C_VEL
LIN {X 0,Y 490.85,Z 635.871,A -85,B 0,C 180,E1 23769.971,E2 23769.971} C_VEL
LIN {X 0,Y 490.403,Z 650.27,A -85,B 0,C 180,E1 23768.855,E2 23768.855} C_VEL
LIN {X 0,Y 489.967,Z 662.833,A -85,B 0,C 180,E1 23767.623,E2 23767.623} C_VEL
LIN {X 0,Y 489.551,Z 674.337,A -85,B 0,C 180,E1 23766.215,E2 23766.215} C_VEL
LIN {X 0,Y 489.189,Z 684.255,A -85,B 0,C 180,E1 23764.69,E2 23764.69} C_VEL
LIN {X 0,Y 488.922,Z 692.72,A -85,B 0,C 180,E1 23763.048,E2 23763.048} C_VEL
LIN {X 0,Y 488.735,Z 699.626,A -85,B 0,C 180,E1 23761.29,E2 23761.29} C_VEL
LIN {X 0,Y 488.619,Z 704.999,A -85,B 0,C 180,E1 23759.414,E2 23759.414} C_VEL
LIN {X 0,Y 488.562,Z 708.571,A -85,B 0,C 180,E1 23757.42,E2 23757.42} C_VEL
LIN {X 0,Y 488.553,Z 710.13,A -85,B 0,C 180,E1 23755.54,E2 23755.54} C_VEL
LIN {X 0,Y 488.597,Z 709.9,A -85,B 0,C 180,E1 23753.538,E2 23753.538} C_VEL
LIN {X 0,Y 488.656,Z 707.81,A -85,B 0,C 180,E1 23751.647,E2 23751.647} C_VEL
LIN {X 0,Y 488.801,Z 703.9,A -85,B 0,C 180,E1 23749.749,E2 23749.749} C_VEL
LIN {X 0,Y 488.958,Z 698.299,A -85,B 0,C 180,E1 23747.961,E2 23747.961} C_VEL
LIN {X 0,Y 489.209,Z 691.212,A -85,B 0,C 180,E1 23746.286,E2 23746.286} C_VEL
LIN {X 0,Y 489.539,Z 681.863,A -85,B 0,C 180,E1 23744.603,E2 23744.603} C_VEL
LIN {X 0,Y 489.908,Z 671.597,A -85,B 0,C 180,E1 23743.154,E2 23743.154} C_VEL
LIN {X 0,Y 490.315,Z 659.717,A -85,B 0,C 180,E1 23741.821,E2 23741.821} C_VEL
LIN {X 0,Y 490.656,Z 647.433,A -85,B 0,C 180,E1 23740.724,E2 23740.724} C_VEL
LIN {X 0,Y 491.011,Z 632.939,A -85,B 0,C 180,E1 23739.706,E2 23739.706} C_VEL
LIN {X 0,Y 491.246,Z 618.335,A -85,B 0,C 180,E1 23738.935,E2 23738.935} C_VEL
LIN {X 0,Y 491.406,Z 602.266,A -85,B 0,C 180,E1 23738.324,E2 23738.324} C_VEL
LIN {X 0,Y 491.413,Z 584.869,A -85,B 0,C 180,E1 23737.92,E2 23737.92} C_VEL
LIN {X 0,Y 492.305,Z 475.107,A -85,B 0,C 180,E1 23736.214,E2 23736.214} C_VEL
LIN {X 0,Y 492.641,Z 450.968,A -85,B 0,C 180,E1 23735.797,E2 23735.797} C_VEL
LIN {X 0,Y 493.151,Z 445.437,A -85,B 0,C 180,E1 23735.377,E2 23735.377} C_VEL
LIN {X 0,Y 493.638,Z 407.116,A -85,B 0,C 180,E1 23732.365,E2 23732.365} C_VEL
LIN {X 0,Y 493.832,Z 373.885,A -85,B 0,C 180,E1 23729.831,E2 23729.831} C_VEL
LIN {X 0,Y 493.641,Z 333.033,A -85,B 0,C 180,E1 23726.847,E2 23726.847} C_VEL
LIN {X 0,Y 493.276,Z 307.194,A -85,B 0,C 180,E1 23725.032,E2 23725.032} C_VEL
LIN {X 0,Y 495.2,Z 308.173,A -85,B 0,C 180,E1 23724.728,E2 23724.728} C_VEL
LIN {X 0,Y 497.547,Z 307.757,A -85,B 0,C 180,E1 23724.496,E2 23724.496} C_VEL
LIN {X 0,Y 499.275,Z 307.112,A -85,B 0,C 180,E1 23724.355,E2 23724.355} C_VEL
LIN {X 0,Y 503.45,Z 306.64,A -85,B 0,C 180,E1 23723.931,E2 23723.931} C_VEL
LIN {X 0,Y 510.268,Z 305.573,A -85,B 0,C 180,E1 23723.284,E2 23723.284} C_VEL
LIN {X 0,Y 508.709,Z 337.957,A -85,B 0,C 180,E1 23720.93,E2 23720.93} C_VEL
LIN {X 0,Y 509.625,Z 353.75,A -85,B 0,C 180,E1 23719.651,E2 23719.651} C_VEL
LIN {X 0,Y 512.199,Z 368.322,A -85,B 0,C 180,E1 23718.342,E2 23718.342} C_VEL
LIN {X 0,Y 516.252,Z 380.735,A -85,B 0,C 180,E1 23717.096,E2 23717.096} C_VEL
LIN {X 0,Y 522.147,Z 392.066,A -85,B 0,C 180,E1 23715.812,E2 23715.812} C_VEL
LIN {X 0,Y 529.363,Z 401.399,A -85,B 0,C 180,E1 23714.596,E2 23714.596} C_VEL
LIN {X 0,Y 537.478,Z 408.817,A -85,B 0,C 180,E1 23713.489,E2 23713.489} C_VEL
LIN {X 0,Y 547.06,Z 415.008,A -85,B 0,C 180,E1 23712.406,E2 23712.406} C_VEL
LIN {X 0,Y 558.154,Z 419.832,A -85,B 0,C 180,E1 23711.36,E2 23711.36} C_VEL
LIN {X 0,Y 563.364,Z 421.315,A -85,B 0,C 180,E1 23710.882,E2 23710.882} C_VEL
LIN {X 0,Y 567.108,Z 421.62,A -85,B 0,C 180,E1 23710.39,E2 23710.39} C_VEL
LIN {X 0,Y 570.025,Z 420.926,A -85,B 0,C 180,E1 23709.801,E2 23709.801} C_VEL
LIN {X 0,Y 571.603,Z 419.227,A -85,B 0,C 180,E1 23709.159,E2 23709.159} C_VEL
LIN {X 0,Y 567.081,Z 432.726,A -85,B 0,C 180,E1 23708.848,E2 23708.848} C_VEL
LIN {X 0,Y 558.953,Z 452.319,A -85,B 0,C 180,E1 23708.762,E2 23708.762} C_VEL
LIN {X 0,Y 549.059,Z 471.558,A -85,B 0,C 180,E1 23708.581,E2 23708.581} C_VEL
LIN {X 0,Y 538.549,Z 489.587,A -85,B 0,C 180,E1 23708.249,E2 23708.249} C_VEL
LIN {X 0,Y 529.692,Z 505.688,A -85,B 0,C 180,E1 23707.773,E2 23707.773} C_VEL
LIN {X 0,Y 524.086,Z 518.715,A -85,B 0,C 180,E1 23707.282,E2 23707.282} C_VEL
LIN {X 0,Y 522.418,Z 522.409,A -85,B 0,C 180,E1 23707.146,E2 23707.146} C_VEL
LIN {X 0,Y 515.711,Z 536.071,A -85,B 0,C 180,E1 23706.666,E2 23706.666} C_VEL
LIN {X 0,Y 507.293,Z 559.843,A -85,B 0,C 180,E1 23705.621,E2 23705.621} C_VEL
LIN {X 0,Y 505.628,Z 566.23,A -85,B 0,C 180,E1 23705.341,E2 23705.341} C_VEL
LIN {X 0,Y 504.799,Z 608.147,A -85,B 0,C 180,E1 23704.661,E2 23704.661} C_VEL
LIN {X 0,Y 503.848,Z 631.268,A -85,B 0,C 180,E1 23704.081,E2 23704.081} C_VEL
LIN {X 0,Y 502.741,Z 652.965,A -85,B 0,C 180,E1 23703.328,E2 23703.328} C_VEL
LIN {X 0,Y 501.518,Z 673.148,A -85,B 0,C 180,E1 23702.432,E2 23702.432} C_VEL
LIN {X 0,Y 500,Z 692.816,A -85,B 0,C 180,E1 23701.328,E2 23701.328} C_VEL
LIN {X 0,Y 498.328,Z 712.606,A -85,B 0,C 180,E1 23699.974,E2 23699.974} C_VEL
LIN {X 0,Y 496.595,Z 731.203,A -85,B 0,C 180,E1 23698.456,E2 23698.456} C_VEL
LIN {X 0,Y 494.841,Z 749.913,A -85,B 0,C 180,E1 23696.652,E2 23696.652} C_VEL
LIN {X 0,Y 493.25,Z 766.685,A -85,B 0,C 180,E1 23694.752,E2 23694.752} C_VEL
LIN {X 0,Y 491.848,Z 782.059,A -85,B 0,C 180,E1 23692.721,E2 23692.721} C_VEL
LIN {X 0,Y 490.644,Z 796.348,A -85,B 0,C 180,E1 23690.519,E2 23690.519} C_VEL
LIN {X 0,Y 489.638,Z 809.739,A -85,B 0,C 180,E1 23688.083,E2 23688.083} C_VEL
LIN {X 0,Y 488.891,Z 821.409,A -85,B 0,C 180,E1 23685.54,E2 23685.54} C_VEL
LIN {X 0,Y 488.407,Z 831.052,A -85,B 0,C 180,E1 23682.979,E2 23682.979} C_VEL
LIN {X 0,Y 488.128,Z 838.895,A -85,B 0,C 180,E1 23680.385,E2 23680.385} C_VEL
LIN {X 0,Y 487.981,Z 844.916,A -85,B 0,C 180,E1 23677.772,E2 23677.772} C_VEL
LIN {X 0,Y 487.927,Z 848.978,A -85,B 0,C 180,E1 23675.291,E2 23675.291} C_VEL
LIN {X 0,Y 487.91,Z 851.571,A -85,B 0,C 180,E1 23672.702,E2 23672.702} C_VEL
LIN {X 0,Y 487.91,Z 852.489,A -85,B 0,C 180,E1 23670.117,E2 23670.117} C_VEL
LIN {X 0,Y 487.909,Z 851.778,A -85,B 0,C 180,E1 23667.651,E2 23667.651} C_VEL
LIN {X 0,Y 487.924,Z 849.589,A -85,B 0,C 180,E1 23665.18,E2 23665.18} C_VEL
LIN {X 0,Y 487.968,Z 845.596,A -85,B 0,C 180,E1 23662.583,E2 23662.583} C_VEL
LIN {X 0,Y 488.091,Z 839.806,A -85,B 0,C 180,E1 23659.972,E2 23659.972} C_VEL
LIN {X 0,Y 488.348,Z 832.527,A -85,B 0,C 180,E1 23657.465,E2 23657.465} C_VEL
LIN {X 0,Y 488.763,Z 823.86,A -85,B 0,C 180,E1 23655.063,E2 23655.063} C_VEL
LIN {X 0,Y 489.435,Z 812.714,A -85,B 0,C 180,E1 23652.524,E2 23652.524} C_VEL
LIN {X 0,Y 490.366,Z 799.914,A -85,B 0,C 180,E1 23650.092,E2 23650.092} C_VEL
LIN {X 0,Y 491.564,Z 785.451,A -85,B 0,C 180,E1 23647.769,E2 23647.769} C_VEL
LIN {X 0,Y 493.023,Z 769.235,A -85,B 0,C 180,E1 23645.561,E2 23645.561} C_VEL
LIN {X 0,Y 494.635,Z 752.047,A -85,B 0,C 180,E1 23643.57,E2 23643.57} C_VEL
